# B&R Automation Studio project Nitto (part 16)

#### FB_GetNextCuttingSynPos.st
```iecst
(********************************************************************
 * COPYRIGHT -- Nitto
 ********************************************************************
 * Programm: MAIN
 * Datei: FB_GetNextCuttingSynPos.st
 * Autor: s_spilker
 * Erstellt: 9. November 2015
 ********************************************************************
 * Implementierung des Programms MAIN
 ********************************************************************)

(* TODO: Bitte Kommentar hier einfügen *)
FUNCTION_BLOCK FB_GetNextCuttingSynPos
// zu brmfmod die Funktion soll einen Rest der zwei Längen berechnen
// wenn die zwei Längen gelich sind (ausgenommen die Nachkommastellen fängt der Wert zu jittern (der Wert springt zwischen 0 und der Periodenlänge)

	periodLength :=	uData.general.periodLength;
	getMark(machineMaster := machineMaster, uData := uData, markpoints := markpoints, uAxis := uAxis, usercorrec := setCutOffset.setOffset_o);
//		IF period = 1 THEN //nur für Testzwecke
//		IF moduloBeforePosition > 0 THEN
//			IF moduloBeforePosition > periodLength THEN
//				correctionTotal1 := fmod(moduloBeforePosition, periodLength);
//				syncDataBefore.correctionNoLimit := correctionTotal1;
//				correctionTotalInt := 1;
//			ELSIF moduloBeforePosition < periodLength THEN
//				syncDataBefore.correctionNoLimit := (periodLength - moduloBeforePosition);
//				correctionTotalInt := 2;
//			END_IF
//		ELSIF 	moduloBeforePosition < 0 THEN
//			IF moduloBeforePosition < - periodLength THEN
//				correctionTotal1 := fmod(moduloBeforePosition, periodLength);
//				syncDataBefore.correctionNoLimit :=  correctionTotal1;
//				correctionTotalInt := 3;
//			ELSIF moduloBeforePosition > - periodLength THEN
//				syncDataBefore.correctionNoLimit := moduloBeforePosition + periodLength;
//				correctionTotalInt := 4;
//			END_IF
//
//		ELSIF moduloBeforePosition = periodLength THEN
//				syncDataBefore.correctionNoLimit := 0;
//				correctionTotalInt := 5;
//		END_IF
//	ELSIF period =	2 THEN
//		IF ABS ( moduloBeforePosition) > periodLength THEN
//			correctionTotal1 := fmod(ABS (moduloBeforePosition), periodLength);
//			syncDataBefore.correctionNoLimit := correctionTotal1 - periodLength;
//			correctionTotalInt := 6;
//		ELSIF ABS (moduloBeforePosition) < periodLength THEN
//			syncDataBefore.correctionNoLimit := correctionTotal1;
//			correctionTotalInt := 7;
//		END_IF
//	ELSIF period = 3 THEN
//			correctionTotal1 := fmod(moduloBeforePosition, periodLength);
//			IF correctionTotal1 > periodLength/2 THEN
//				syncDataBefore.correctionNoLimit := correctionTotal1 - periodLength;
//			ELSE
//				syncDataBefore.correctionNoLimit := correctionTotal1;
//			END_IF
//	ELSIF period =4 THEN
//			correctionTotal1 := fmod(ABS (moduloBeforePosition), periodLength);
//				IF correctionTotal1 > periodLength/2 THEN
//				syncDataBefore.correctionNoLimit := correctionTotal1 - periodLength;
//			ELSE
//				syncDataBefore.correctionNoLimit := correctionTotal1;
//			END_IF
//	ELSIF period = 5 THEN
//		correctionTotal1 := fmod(moduloBeforePosition, periodLength);
//	END_IF
//////permantes Lesen der Kurvenscheibenposition des Masters X-Achse 607, 512, 1067,
//	MC_BR_ReadCyclicPosition_1(Enable := TRUE, ParID:= 542, Axis := uAxis.AxisREF);//nur zu Testzwecken
	MC_BR_ReadCyclicPosition_0(Enable := TRUE, ParID:= 1075, Axis := uAxis.AxisREF);
//	moduloBeforePosition := MC_BR_ReadCyclicPosition_0.CyclicPosition.Integer - uData.general.periodLength;
	moduloBeforePosition := MC_BR_ReadCyclicPosition_0.CyclicPosition.Real - uData.general.periodLength;
	IF uData.recipe.mode = CONST.CUTTINGUNIT.MODEs.FREE_RUN THEN
		//für einen Rundenzähler
		countRtrig();
		IF MC_BR_ReadCyclicPosition_0.CyclicPosition.Real < 5000 THEN
			countRtrig.CLK := TRUE;
		END_IF
		IF countRtrig.Q	THEN
			syncDataBefore.markIndx := syncDataBefore.markIndx + 1;
			syncDataBefore.correctionNoLimit :=	- setCutOffset.setOffset_o;
		END_IF
		IF MC_BR_ReadCyclicPosition_0.CyclicPosition.Real > 10000 THEN
			countRtrig.CLK := FALSE;
		END_IF
	ELSIF uData.recipe.mode = CONST.CUTTINGUNIT.MODEs.SYNC_RUN OR uData.recipe.mode = CONST.CUTTINGUNIT.MODEs.CROSS_CUT THEN
			IF 	markpoints.ProbeCounter <> tmpcounter  OR trigger THEN
	//			correctionTotal := getMark.diffToUnitBefore - MC_BR_ReadCyclicPosition_0.CyclicPosition.Real;
				correctionTmp	:= fmod(getMark.diffToUnitBefore, uData.general.periodLength);
	//			correctionTotal := getMark.diffToUnitBefore - moduloBeforePosition;////03.11
				correctionTotal := correctionTmp - moduloBeforePosition;
				syncDataBefore.correctionNoLimit := correctionTotal;
				trigger := FALSE;
				syncDataBefore.markIndx := markpoints.ProbeCounter;
				tmpcounter := markpoints.ProbeCounter;
			ELSIF markpoints.MissedTriggers <> period THEN
				syncDataBefore.correctionNoLimit := correctionTotal;// LETZTEN BEKQNNTN WERT ALS KORREKTUR VORGEBEN
				period := markpoints.MissedTriggers;
			END_IF
	END_IF

END_FUNCTION_BLOCK
```

#### FB_CreateCamTable.st
```iecst
(********************************************************************
 * COPYRIGHT -- Nitto
 ********************************************************************
 * Programm: MAIN
 * Datei: FB_CreateCamTable.st
 * Autor: s_spilker
 * Erstellt: 9. November 2015
 ********************************************************************
 * Implementierung des Programms MAIN
 ********************************************************************)

(* TODO: Bitte Kommentar hier einfügen *)
FUNCTION_BLOCK FB_CreateCamTable
	CASE state OF

		STATE_READY://0
			IF createCam THEN
				(*	createCam:=FALSE;*)
				err(reset := TRUE);
				IF  data.recipe.tool.numberToolSegments = 1 OR data.recipe.tool.numberToolSegments = 0 OR data.recipe.mode = CONST.CUTTINGUNIT.MODEs.FREE_RUN THEN
					idx := 0;
					state:=STATE_CALCULATE_CAM1;
				ELSIF data.recipe.tool.numberToolSegments > 1 AND data.recipe.mode = CONST.CUTTINGUNIT.MODEs.SYNC_RUN THEN
					idx := 0;
					jdx := 0;
					state:=STATE_CALCULATE_CAM2;
				END_IF
			ELSE
				done:=FALSE;
			END_IF
		(*********************************************)
		STATE_CALCULATE_CAM1://1  (*calculate cam from sections*)
			(*bestimmung der Eigenschaften der Stützpunkte. Es können bis zu 64 Stützpunkte angelegt werden*)
			IF data.recipe.mode = CONST.CUTTINGUNIT.MODEs.FREE_RUN THEN // beim Freilauf wird Insetting auf ganzen Umfang bezogen
				CamSections.Section[0].MasterPosition	:=0;
				CamSections.Section[0].SlavePosition	:=0;
				CamSections.Section[0].FirstDerivative 	:= 1; (* Laut Ronny bei 1 wird die Geschwind. vom Master übernommen'*)
				CamSections.Section[0].SecondDerivative := 0;
				CamSections.Section[0].Mode 			:= mcABSOLUTE;(*mcRELATIVE;*)
				CamSections.Section[0].Type 			:= mc5TH_ORDER_POLYNOMIAL;

				CamSections.Section[1].MasterPosition 	:= scalePerimeter.realperimeter;// da das Werkzeug 1 zu 1 laufen soll
				CamSections.Section[1].SlavePosition 	:= scalePerimeter.realperimeter;
				CamSections.Section[1].FirstDerivative 	:= 1;
				CamSections.Section[1].SecondDerivative	:= 0;
				CamSections.Section[1].Mode 			:= mcABSOLUTE;  (*mcRELATIVE;*)
				CamSections.Section[1].Type 			:= mcLAST_POINT;(* mc5TH_ORDER_POLYNOMIAL;*)
				idx := 2;
				maxIdx := 64;
				WHILE idx < maxIdx -1 DO // falls bereits Stützpunkte vorhanden, alle löschen
					CamSections.Section[idx].MasterPosition		:= 0;
					CamSections.Section[idx].SlavePosition 		:= 0;
					CamSections.Section[idx].FirstDerivative 	:= 0; (* Laut Ronny bei 1 wird die Geschwind. vom Master übernommen'*)
					CamSections.Section[idx].SecondDerivative 	:= 0;
					CamSections.Section[idx].Mode 				:= 0;
					CamSections.Section[idx].Type 				:= 0;///mc5TH_ORDER_POLYNOMIAL;
					idx := idx +1;
				END_WHILE

				state:= STATE_CALC_CAM_FROM_SECTIONS;

			ELSIF data.recipe.mode = CONST.CUTTINGUNIT.MODEs.SYNC_RUN OR data.recipe.mode = CONST.CUTTINGUNIT.MODEs.CROSS_CUT THEN

				IF   data.recipe.tool.cutEndPosition > data.recipe.tool.cutStartPosition AND data.recipe.tool.cutEndPosition > 0 THEN
					//Kurvenscheibe mit einer synchnoner Strecke
					CamSections.Section[0].MasterPosition:=0;
					CamSections.Section[0].SlavePosition:=0;
					CamSections.Section[0].FirstDerivative := 1; (* Laut Ronny bei 1 wird die Geschwind. vom Master übernommen'*)
					CamSections.Section[0].SecondDerivative := 0;
					CamSections.Section[0].Mode := mcABSOLUTE;(*mcRELATIVE;*)
					CamSections.Section[0].Type := mcSTRAIGHT_LINE;///mc5TH_ORDER_POLYNOMIAL;
					// Ende der Kurvenscheibenstrecke mit einem automatischen Ausgleich und Anfang des Ausgleichs
					CamSections.Section[1].MasterPosition:= data.recipe.tool.cutEndPosition;
					CamSections.Section[1].SlavePosition:=data.recipe.tool.cutEndPosition;
					CamSections.Section[1].FirstDerivative := 1; (* Laut Ronny bei 1 wird die Geschwind. vom Master übernommen'*)
					CamSections.Section[1].SecondDerivative := 0;
					CamSections.Section[1].Mode := mcABSOLUTE;(*mcRELATIVE;*)
					CamSections.Section[1].Type := mc5TH_ORDER_POLYNOMIAL;//mcHARMONIC_COMBINATION ;
					//
					CamSections.Section[2].MasterPosition :=data.general.periodLength;
					CamSections.Section[2].SlavePosition := scalePerimeter.realperimeter;
					CamSections.Section[2].FirstDerivative := 1;
					CamSections.Section[2].SecondDerivative:= 0;
					CamSections.Section[2].Mode := mcABSOLUTE;  (*mcRELATIVE;*)
					CamSections.Section[2].Type := mcLAST_POINT;(* mc5TH_ORDER_POLYNOMIAL;*)

					idx := 3;
					maxIdx := 64;
					WHILE idx < maxIdx -1 DO // falls bereits Stützpunkte vorhanden, alle löschen

						CamSections.Section[idx].MasterPosition		:= 0;
						CamSections.Section[idx].SlavePosition 		:= 0;
						CamSections.Section[idx].FirstDerivative 	:= 0; (* Laut Ronny bei 1 wird die Geschwind. vom Master übernommen'*)
						CamSections.Section[idx].SecondDerivative 	:= 0;
						CamSections.Section[idx].Mode 				:= 0;
						CamSections.Section[idx].Type 				:= 0;///mc5TH_ORDER_POLYNOMIAL;
						idx := idx +1;
					END_WHILE
					state:= STATE_CALC_CAM_FROM_SECTIONS;

				ELSIF  data.recipe.tool.cutEndPosition = 0 OR data.recipe.tool.cutEndPosition = scalePerimeter.realperimeter THEN
					CamSections.Section[0].MasterPosition:=0;
					CamSections.Section[0].SlavePosition:=0;
					CamSections.Section[0].FirstDerivative := 1; (* Laut Ronny bei 1 wird die Geschwind. vom Master übernommen'*)
					CamSections.Section[0].SecondDerivative := 0;
					CamSections.Section[0].Mode := mcABSOLUTE;(*mcRELATIVE;*)
					CamSections.Section[0].Type := mc5TH_ORDER_POLYNOMIAL;

					CamSections.Section[1].MasterPosition :=data.general.periodLength;
					CamSections.Section[1].SlavePosition := scalePerimeter.realperimeter;
					CamSections.Section[1].FirstDerivative := 1;
					CamSections.Section[1].SecondDerivative:= 0;
					CamSections.Section[1].Mode := mcABSOLUTE;  (*mcRELATIVE;*)
					CamSections.Section[1].Type := mcLAST_POINT;(* mc5TH_ORDER_POLYNOMIAL;*)
					idx := 2;
					maxIdx := 64;
					WHILE idx < maxIdx -1 DO // falls bereits Stützpunkte vorhanden, alle löschen
						CamSections.Section[idx].MasterPosition		:= 0;
						CamSections.Section[idx].SlavePosition 		:= 0;
						CamSections.Section[idx].FirstDerivative 	:= 0; (* Laut Ronny bei 1 wird die Geschwind. vom Master übernommen'*)
						CamSections.Section[idx].SecondDerivative 	:= 0;
						CamSections.Section[idx].Mode 				:= 0;
						CamSections.Section[idx].Type 				:= 0;///mc5TH_ORDER_POLYNOMIAL;
						idx := idx +1;
					END_WHILE
					state:= STATE_CALC_CAM_FROM_SECTIONS;
				END_IF
			ELSIF data.recipe.tool.cutEndPosition < data.recipe.tool.cutStartPosition THEN
				err.set := TRUE;
				err.state := state;
				err.text := 'Synchronerbereich ist größer als Nutzen';
				err.fnc := 'FB_Camtable';
				err.id := MC_BR_CalcCamFromSections_0.ErrorID;
				state:=STATE_ERROR;
			END_IF

		STATE_CALCULATE_CAM2://1  (*calculate cam from sections*)
			(*Bestimmung der Eigenschaften der Stützpunkte. Es können bis zu 64 Stützpunkte angelegt werden*)
			IF data.recipe.tool.numberToolSegments > 1 AND  data.recipe.tool.numberToolSegments <= 12 THEN
				partOfPerimeter := scalePerimeter.realperimeter/data.recipe.tool.numberToolSegments;  //Anzahl der Kurvenstücken
				maxIdx			:= data.recipe.tool.numberToolSegments *2;
			ELSE
				partOfPerimeter := scalePerimeter.realperimeter;
			END_IF

			IF data.recipe.tool.cutEndPosition < partOfPerimeter  THEN
				CamSections.Section[maxIdx].MasterPosition	:= scalePerimeter.realperimeter;
				CamSections.Section[maxIdx].SlavePosition	:= scalePerimeter.realperimeter;
				CamSections.Section[maxIdx].FirstDerivative := 1; (* Laut Ronny bei 1 wird die Geschwind. vom Master übernommen'*)
				CamSections.Section[maxIdx].SecondDerivative:= 0;
				CamSections.Section[maxIdx].Mode 			:= mcABSOLUTE;
				CamSections.Section[maxIdx].Type 			:= mcLAST_POINT;
				WHILE idx < maxIdx -1 DO //jeden zweiten Stützpunkt, gerade Zahl
					CamSections.Section[idx].MasterPosition		:= partOfPerimeter * jdx;
					CamSections.Section[idx].SlavePosition 		:= partOfPerimeter * jdx;
					CamSections.Section[idx].FirstDerivative 	:= 1;
					CamSections.Section[idx].SecondDerivative 	:= 0;
					CamSections.Section[idx].Mode 				:= mcABSOLUTE;
					CamSections.Section[idx].Type 				:= mcSTRAIGHT_LINE; //mc5TH_ORDER_POLYNOMIAL;
					idx := idx + 2;
					jdx := jdx + 1;
				END_WHILE

				idx := 1;
				jdx := 0;
				WHILE idx < maxIdx DO//jede ungeraden Stützpuknt
					CamSections.Section[idx].MasterPosition		:= partOfPerimeter * jdx + data.recipe.tool.cutEndPosition;
					CamSections.Section[idx].SlavePosition 		:= partOfPerimeter * jdx + data.recipe.tool.cutEndPosition;
					CamSections.Section[idx].FirstDerivative 	:= 1; (* Laut Ronny bei 1 wird die Geschwind. vom Master übernommen'*)
					CamSections.Section[idx].SecondDerivative 	:= 0;
					CamSections.Section[idx].Mode 				:= mcABSOLUTE;
					CamSections.Section[idx].Type 				:= mc5TH_ORDER_POLYNOMIAL;///
					idx := idx + 2;
					jdx := jdx + 1;
				END_WHILE
				state:= STATE_CALC_CAM_FROM_SECTIONS;
			ELSE
				err.set := TRUE;
				err.state := state;
				err.text := 'Synchronerbereich ist größer als Nutzen';
				err.fnc := 'FB_Camtable';
				err.id := MC_BR_CalcCamFromSections_0.ErrorID;
				state:=STATE_ERROR;
			END_IF

		STATE_CALC_CAM_FROM_SECTIONS://2 //hier werden einzelne Punkte die in STATE_CALCULATE_CAM angelegt wurden sind als eine Stätige Kurve zusammen gesetzt
			idx := 0;
			MC_BR_CalcCamFromSections_0.Execute:= TRUE;
			MC_BR_CalcCamFromSections_0.DataAddress:=ADR(CamSections);
			MC_BR_CalcCamFromSections_0.CamProfileAddress:=ADR(MC_CAMPROFILE_TYP_0);
			MC_BR_CalcCamFromSections_0();

			IF MC_BR_CalcCamFromSections_0.Done THEN
				MC_BR_CalcCamFromSections_0.Execute:= FALSE;
				(*state:=STATE_READY;*)
				state := STATE_SAVE_CAM_PROFILE;
			ELSIF MC_BR_CalcCamFromSections_0.Error THEN
				err.set := TRUE;
				err.state:= state;
				err.text :='MC_BR_CalcCamFromSections_0';
				err.fnc := 'FB_Camtable';
				err.id := MC_BR_CalcCamFromSections_0.ErrorID;
				axis1ErrorID:= MC_BR_CalcCamFromSections_0.ErrorID;
				MC_BR_CalcCamFromSections_0.Execute:=0;
				state:=STATE_ERROR;
			END_IF

		STATE_SAVE_CAM_PROFILE:  //3 schreibe die Kurvenscheibe in das NC-Kurvenscheiben-Datenmodul
			MC_BR_CalcCamFromSections_0(); //noch einen Zyklus aufrufen

			MC_BR_SaveCamProfileObj_0.Execute			:= TRUE;
			MC_BR_SaveCamProfileObj_0.DataObjectName	:= Name; //'TestCam'; //Sehr wichtig der Name darf nicht größer als 12 Zeichen sein
			// Wie es bei B&R üblich ist, steht es explizit nirgendswo geschrieben. Nach mühsamen Test hat sich es gezeigt.
			MC_BR_SaveCamProfileObj_0.DataAddress		:= ADR(MC_CAMPROFILE_TYP_0);
			MC_BR_SaveCamProfileObj_0.DataObjectVersion	:= 1000;

			MC_BR_SaveCamProfileObj_0();

			IF MC_BR_SaveCamProfileObj_0.Done  THEN
				MC_BR_SaveCamProfileObj_0.Execute	:= FALSE;
				state:=STATE_DOWNLOAD_CAMPROFILEDATA;
			ELSIF MC_BR_SaveCamProfileObj_0.Error THEN
				err.set := TRUE;
				err.state := state;
				err.text := 'MC_BR_SaveCamProfileObj_0';
				err.fnc := 'FB_Camtable';
				err.id := MC_BR_SaveCamProfileObj_0.ErrorID;
				state := STATE_ERROR;
			END_IF

		STATE_DOWNLOAD_CAMPROFILEDATA://4 übertrage die Daten vom NC-Kurvenscheiben-Datenmodul auf den Antrieb
			(* zulässiger  an index for cam (1-14)*)
			MC_BR_SaveCamProfileObj_0();

			MC_BR_DownloadCamProfileObj_0.Execute 		:= TRUE;
			MC_BR_DownloadCamProfileObj_0.DataObjectName:= Name;
			MC_BR_DownloadCamProfileObj_0.Index			:= index;
			MC_BR_DownloadCamProfileObj_0.Periodic		:= mcPERIODIC;

			MC_BR_DownloadCamProfileObj_0(Axis := AxisREF);

			IF MC_BR_DownloadCamProfileObj_0.Done THEN
				MC_BR_DownloadCamProfileObj_0.Execute := FALSE;
				state :=  STATE_CAMTABLE_SEL;
			ELSIF MC_BR_DownloadCamProfileObj_0.Error THEN
				err.set := TRUE;
				err.state :=  state;
				err.text := 'MC_BR_DownloadCamProfileObj_0';
				err.fnc := 'FB_Camtable';
				err.id := MC_BR_DownloadCamProfileObj_0.ErrorID;
				state := STATE_ERROR;
			END_IF

		STATE_CAMTABLE_SEL: //5 wählt eine vordefinierte Kurvensscheibe ausfür den FB MC_CamIn.
			MC_BR_DownloadCamProfileObj_0(Axis := AxisREF);

			MC_CamTableSelect_0.CamTable := Name;
			MC_CamTableSelect_0.Periodic := mcPERIODIC; //periodische Achse
			MC_CamTableSelect_0.Execute := TRUE;
			MC_CamTableSelect_0(Master := MasterAxisREF, Slave := AxisREF);
			IF MC_CamTableSelect_0.Done AND MC_CamTableSelect_0.CamTableID > 0 THEN
				camTableID := MC_CamTableSelect_0.CamTableID; //zwischenspeichern weil beim nächsten Aufruf die CamTableID auf 0 gesetzt wird
				MC_CamTableSelect_0.Execute := FALSE;
				(*	done:=TRUE;*)
				//	createCam:=FALSE;//16.04.15 wird aus dem Config auf rückgesetzt.
				state := STATE_COMPLETED;
			ELSIF MC_CamTableSelect_0.Error THEN
				err(set := TRUE, text := 'MC_CamTableSelect_0', fnc := 'FB_Camtable', id := MC_CamTableSelect_0.ErrorID);
				state := STATE_ERROR;
			END_IF

		STATE_COMPLETED://10 FB werden noch mal aufgerufen um den Ausgang Done auf false zu setzten
			MC_BR_CalcCamFromSections_0(Execute := FALSE);
			MC_BR_SaveCamProfileObj_0(Execute := FALSE);
			MC_BR_DownloadCamProfileObj_0(Execute := FALSE);
			MC_CamTableSelect_0(Master := MasterAxisREF, Slave := AxisREF, Execute := FALSE);
			IF data.recipe.mode = CONST.CUTTINGUNIT.MODEs.FREE_RUN THEN
				IF MC_CAMPROFILE_TYP_0.MasterPeriod = REAL_TO_DINT(scalePerimeter.realperimeter) AND MC_CAMPROFILE_TYP_0.SlavePeriod = REAL_TO_DINT (scalePerimeter.realperimeter) THEN
					done:=TRUE;
					state := STATE_READY;
				END_IF
			ELSIF data.recipe.mode = CONST.CUTTINGUNIT.MODEs.SYNC_RUN THEN
				IF (*MC_CAMPROFILE_TYP_0.MasterPeriod >= REAL_TO_DINT(scalePerimeter.realperimeter) AND *)MC_CAMPROFILE_TYP_0.SlavePeriod = REAL_TO_DINT (scalePerimeter.realperimeter) THEN
					done:=TRUE;
					state := STATE_READY;
				END_IF
			END_IF

		STATE_ERROR:
			createCam:=FALSE;
			err();
			state:=STATE_READY;

	END_CASE
END_FUNCTION_BLOCK
```

#### FB_MARK_POSITION.st
```iecst
(********************************************************************
 * COPYRIGHT -- Nitto
 ********************************************************************
 * Programm: MAIN
 * Datei: FB_MARK_POSITION.st
 * Autor: s_spilker
 * Erstellt: 9. November 2015
 ********************************************************************
 * Implementierung des Programms MAIN
 ********************************************************************)

(* TODO: Bitte Kommentar hier einfügen *)
FUNCTION_BLOCK FB_MARK_POSITION
END_FUNCTION_BLOCK
```

#### Package Logical/MainMachineCtrl/MAIN/Longcutter - Paket

#### ac_manualLongCut.st
```iecst
(********************************************************************
 * COPYRIGHT -- Microsoft
 ********************************************************************
 * Programm: MAIN
 * Datei: acmanualLongCut.st
 * Autor: awalz
 * Erstellt: 30. Juni 2014
 ********************************************************************
 * Implementierung des Programms MAIN
 ********************************************************************)

(* Fügt eine neue Aktion zum IEC Programm oder Bibliothek *)
ACTION ac_manualLongCut:
		axis.ctrl();
		config( machineMasterCtrl := machineMaster, axis := axis, status := status);
	CASE state OF
	ST_IDLE:
		IF config.busy OR config.cmd <> CONST.CUTTINGUNIT.CMDs.NO_CMD THEN
			config(cmd := CONST.CUTTINGUNIT.CMDs.NO_CMD, machineMasterCtrl := machineMaster, axis := axis, status := status);
		ELSIF manualFirst  OR mode <> status.mode (*OR NewData *)THEN
			IF NOT status.isCoupled AND mode = CONST.UNITMODEs.ENABLE (*AND axis.ctrl.MC_ReadStatus_0.Disabled *)THEN
				axis.ctrl(cmd:= CONST.AXIS.POWER_ON);
				IF axis.ctrl.MC_ReadStatus_0.StandStill THEN
					status(mode := mode,axisState := axis.ctrl.MC_ReadStatus_0 );
					config(cmd := CONST.CUTTINGUNIT.CMDs.CPL_ON, machineMasterCtrl := machineMaster, axis := axis, status := status);
					state := ST_CPL_WAIT;
				END_IF
			ELSIF mode = CONST.UNITMODEs.DISABLE AND status.isCoupled THEN
				status(mode := mode,axisState := axis.ctrl.MC_ReadStatus_0 );
				config(cmd := CONST.CUTTINGUNIT.CMDs.CPL_OFF, machineMasterCtrl := machineMaster, axis := axis, status := status);
				state := ST_CPL_WAIT;
//			ELSIF	mode = CONST.UNITMODEs.AXIS_OFF THEN
//				status(mode := mode,axisState := axis.ctrl.MC_ReadStatus_0 );
//				axis.ctrl(cmd:= CONST.AXIS.POWER_OFF);
//				status.isCoupled := FALSE;
//				state := ST_AXIS_OFF;
//			ELSIF	mode = CONST.UNITMODEs.DISABLE AND axis.ctrl.MC_ReadStatus_0.Disabled THEN
//				status(mode := mode,axisState := axis.ctrl.MC_ReadStatus_0 );
//				status.isCoupled := FALSE;
//				axis.ctrl(cmd:= CONST.AXIS.POWER_ON);
//				state := ST_AXIS_ON;
////////////////////////
			ELSIF cmdCtrl.value = CONST.CUTTINGUNIT.CMDs.MOVEFW (*OR cmdCtrl.value = CONST.CUTTINGUNIT.CMDs.MOVEBW*) THEN
				cmdStatus(set := TRUE, value := cmdCtrl.value);
				busy := TRUE;
				state := ST_MOVE_START;
//////////////////////////
			ELSE
				NewData := FALSE;
				manualFirst := FALSE;
			END_IF
		ELSIF cmdCtrl.value <> CONST.CUTTINGUNIT.CMDs.NO_CMD THEN
			cmdStatus(set := TRUE, value := cmdCtrl.value);
			busy := TRUE;
			state := ST_FUNCTION_START;
		END_IF

	ST_CPL_WAIT:
		config( machineMasterCtrl := machineMaster, axis := axis, status := status);
		(*status(mode := mode);*)
		IF NOT config.busy THEN
			IF config.err.flag THEN
				err := config.err;
				err.state := state;
				state := ST_ERROR;
			ELSE
				manualFirst := FALSE;
				axis.setGearRatio.init := TRUE;  // OKrebs 09.12.15
				state := ST_IDLE;
			END_IF
			config(cmd := CONST.CUTTINGUNIT.CMDs.NO_CMD, machineMasterCtrl := machineMaster, axis := axis, status := status );
		END_IF

	ST_FUNCTION_START:
		IF config.busy OR config.cmd <> CONST.CUTTINGUNIT.CMDs.NO_CMD THEN
			config(cmd := CONST.CUTTINGUNIT.CMDs.NO_CMD, machineMasterCtrl := machineMaster, axis := axis, status := status);
		ELSE
			config(cmd := cmdStatus.value, machineMasterCtrl := machineMaster, axis := axis, status := status);
			state := ST_FUNCTION;
		END_IF

	ST_FUNCTION:
		config( machineMasterCtrl := machineMaster, axis := axis, status := status);
		IF NOT config.busy THEN
			IF config.err.flag THEN
				err := config.err;
				err.state := state;
			END_IF
			config(cmd := CONST.CUTTINGUNIT.CMDs.NO_CMD, machineMasterCtrl := machineMaster, axis := axis, status := status );
			state := ST_FUNCTION_QUIT;
		END_IF
////12.08.14/////
	ST_MOVE_START:
			config(cmd := cmdStatus.value, machineMasterCtrl  := machineMaster, axis := axis, status := status);
			state := ST_MOVE;

	ST_MOVE:
//		config (machineMaster := machineMaster, axis := axis, status := status, data := data, IOs := IOs, powerbridge := powerbridge,
//				scalePerimeter := scalePerimeter, getNextCuttPos := getNextCuttPos);
		IF cmdCtrl.value = CONST.CUTTINGUNIT.CMDs.NO_CMD THEN
			config(cmd := CONST.CUTTINGUNIT.CMDs.NO_CMD, machineMasterCtrl := machineMaster, axis := axis, status := status);
			state := ST_MOVE_QUIT;

		ELSE
			config(cmd := cmdStatus.value, machineMasterCtrl := machineMaster, axis := axis, status := status);
		END_IF

	ST_MOVE_QUIT:
		config(cmd := CONST.CUTTINGUNIT.CMDs.NO_CMD, machineMasterCtrl := machineMaster, axis := axis, status := status);
		IF NOT config.busy THEN
			busy := FALSE;
			cmdStatus(set := TRUE, value := CONST.CUTTINGUNIT.CMDs.NO_CMD);
			state := ST_IDLE;
		END_IF

////////////////////////////////
	ST_AXIS_OFF:
	(*	status(mode := mode);*)
		IF mode <> CONST.UNITMODEs.AXIS_OFF THEN
			state := ST_IDLE;
		END_IF
	ST_AXIS_ON:
	(*	status(mode := mode);*)
		IF mode <> CONST.UNITMODEs.DISABLE THEN
			state := ST_IDLE;
		END_IF

	ST_FUNCTION_QUIT:
		busy := FALSE;
		IF cmdCtrl.value = CONST.CUTTINGUNIT.CMDs.NO_CMD THEN
			cmdStatus(set :=TRUE, value := CONST.CUTTINGUNIT.CMDs.NO_CMD);
			state := ST_IDLE;
		END_IF

	ST_ERROR:
		err.flag := TRUE;
		busy := FALSE;
		IF BetrCtrl.value <> CONST.MACHINEMODES.MANUAL THEN
			state := ST_IDLE;
			err(reset := TRUE);
			busy := TRUE;
			StateCtrl := CTRL_MANUAL_AFTER;
		END_IF
	END_CASE

	(*axis.calcGearRatio(enable := ( data.torqueCtrlOn  AND axis.ctrl.ref.Status.Coupled), axisRef := axis.ctrl.ref, zugRegelWert := zugRegelWert);*)
END_ACTION
```

#### FB_LongcutterCtrl.st
```iecst
(********************************************************************
 * COPYRIGHT -- Microsoft
 ********************************************************************
 * Programm: MAIN
 * Datei: FB_LongcutterCtrl.st
 * Autor: awalz
 * Erstellt: 29. Juni 2014
 ********************************************************************
 * Implementierung des Programms MAIN
 ********************************************************************)

(* TODO: Bitte Kommentar hier einfügen *)
FUNCTION_BLOCK FB_LongcutterCtrl
	axis.ctrl();
	cutterUp(clk := clk, );(*cutterUp.enable wird dierekt vom EIngang 202A3Input6 geschaltet*)
	discmovesupp(clk := clk);
	movebutton(clk := clk);
	webclamp(clk := clk);
	status(axisState := axis.ctrl.MC_ReadStatus_0);
	status.ready := axis.ctrl.MC_ReadStatus_0.SynchronizedMotion;
	emcy_inputs();
	IF emcy_inputs.EMCY_Door1 THEN
		emcy_inputs.EMCY_DoorsClosed := TRUE;
	ELSE
		emcy_inputs.EMCY_DoorsClosed := FALSE;

	END_IF
	chkStatus(setMode := mode, status := status);
	axis.setGearRatio(limitvisuneg := -20, limitvisupos := 50, limitrationeg := 800, limitratiopos := 1500);
	IF machineMaster.MC_ReadStatus_0.ContinuousMotion THEN
		discmovesupp.toDown_o := FALSE;
	END_IF
//	IF axis.ctrl.MC_ReadStatus_0.SynchronizedMotion AND axis.setGearRatio.enable THEN
//
//
//	END_IF
	axis.cplOn.Execute := axis.setGearRatio.trigger OR movebutton.LDT.ftrig.Q OR axisCpl; // 25.07.18 // OKrebs

	axis.cplOn(RatioNumerator := axis.setGearRatio.ratioNumeratorOut,
				(*Execute := axis.setGearRatio.trigger, 25.07.18 OKrebs*) RatioDenominator := axis.setGearRatio.ratioDenominator,
					Acceleration := 40000, Deceleration := 40000);

//	IF  movebutton.LDT.ftrig.Q THEN	// 25.07.18 // OKrebs
//		axis.cplOn.Execute := TRUE; // 25.07.18 // OKrebs
//	END_IF							// 25.07.18 // OKrebs

////12.08.14 jog set commando  for Longcutter
	IF movebutton.LDT.button THEN
		cmdCtrl.value := CONST.CUTTINGUNIT.CMDs.MOVEFW;
	ELSIF movebutton.LDT.ftrig.Q THEN ////12.08.14 jog reset commando  for Longcutter
		cmdCtrl.value := CONST.CUTTINGUNIT.CMDs.NO_CMD;
	END_IF
////21.08.14 Um Achse zu reseten//
	IF cmdCtrl.value = CONST.CUTTINGUNIT.CMDs.RESET THEN
		axis.ctrl.cmd := CONST.AXIS.RESET;
	ELSIF cmdCtrl.value = CONST.CUTTINGUNIT.CMDs.NO_CMD THEN
		axis.ctrl.cmd := CONST.AXIS.NOACTION;
	END_IF
	status.axiserror := axis.ctrl.MC_ReadStatus_0.Errorstop;
	IF	mode = CONST.UNITMODEs.AXIS_OFF OR  NOT emcy_inputs.EMCY_Door1 THEN
				status(mode := mode,axisState := axis.ctrl.MC_ReadStatus_0 );
				axis.ctrl(cmd:= CONST.AXIS.POWER_OFF);
				status.isCoupled := FALSE;
				state := ST_AXIS_OFF;
	ELSIF	mode = CONST.UNITMODEs.ENABLE AND axis.ctrl.MC_ReadStatus_0.Disabled AND  emcy_inputs.EMCY_Door1 THEN
				status(mode := mode,axisState := axis.ctrl.MC_ReadStatus_0 );
				status.isCoupled := FALSE;
				axis.ctrl(cmd:= CONST.AXIS.POWER_ON);
				stateCPL := cpl_idle;
	ELSIF	mode = CONST.UNITMODEs.DISABLE AND NOT axis.ctrl.MC_ReadStatus_0.Disabled AND  emcy_inputs.EMCY_Door1 THEN
				status(mode := mode,axisState := axis.ctrl.MC_ReadStatus_0 );
				status.isCoupled := FALSE;
				axis.ctrl(cmd:= CONST.AXIS.POWER_ON);
				state := ST_AXIS_ON;
	END_IF
//////////////////////
	CASE stateCPL OF
		cpl_idle :
			IF axis.ctrl.MC_ReadStatus_0.StandStill THEN
				axisCpl := TRUE;
//				axis.cplOn.Execute := TRUE; // 25.07.18 // OKrebs
				stateCPL := clp_cpl;
			END_IF
		clp_cpl:
			axisCpl := FALSE;
				;
		END_CASE
	CASE StateCtrl OF
	CTRL_FIRST_START:
		busy := TRUE;
		StateCtrl := CTRL_EMERGENCYSTOP_BEFORE;

	CTRL_MANUAL_BEFORE:
		IF BetrCtrl.value = CONST.MACHINEMODES.MANUAL THEN
		(*	clamp.init(clk := clk);*)
			BetrStatus(set := TRUE, value := CONST.MACHINEMODES.MANUAL);
			chkStatus.enable := TRUE;
			err(reset := TRUE);
			busy := FALSE;
			timer(IN:= FALSE);
			state := ST_IDLE;
			manualFirst := TRUE;
			StateCtrl := CTRL_MANUAL;
//			axis.setGearRatio.init := TRUE;
		ELSIF BetrCtrl.value = CONST.MACHINEMODES.EMERGENCYSTOP THEN
			StateCtrl := CTRL_EMERGENCYSTOP_BEFORE;
		ELSIF BetrCtrl.value = CONST.MACHINEMODES.SAFETYSTOP THEN
			StateCtrl := CTRL_SAFETYSTOP_BEFORE;
		ELSIF BetrCtrl.value = CONST.MACHINEMODES.AUTOMATIC THEN
			StateCtrl := CTRL_AUTO_BEFORE;
		END_IF

	CTRL_MANUAL:
		IF BetrCtrl.value <> CONST.MACHINEMODES.MANUAL THEN
			err(reset := TRUE);
			busy := TRUE;
			StateCtrl := CTRL_MANUAL_AFTER;
//		ELSIF axis.ctrl.MC_ReadStatus_0.StandStill THEN
//			axis.ctrl.cmd := CONST.AXIS.START;
//				timer(IN := TRUE, PT := T#8s);
//				IF timer.Q THEN

			(*	END_IF*)
		ELSE
			ac_manualLongCut;
		END_IF

	CTRL_MANUAL_AFTER:
		timer(IN:= FALSE);
		chkStatus.enable := FALSE;
		axis.ctrl.cmd := CONST.AXIS.NOACTION;
		ac_setStateAfterPB;

	CTRL_AUTO_BEFORE:
		IF BetrCtrl.value = CONST.MACHINEMODES.AUTOMATIC THEN
		BetrStatus(set := TRUE, value := CONST.MACHINEMODES.AUTOMATIC);
			(*clamp.init(clk := clk);*)
			err(reset := TRUE);
			chkStatus.enable := TRUE;
			busy := FALSE;
			state := ST_IDLE;
			StateCtrl := CTRL_AUTO;
		ELSIF BetrCtrl.value = CONST.MACHINEMODES.EMERGENCYSTOP THEN
			StateCtrl := CTRL_EMERGENCYSTOP_BEFORE;
		ELSIF BetrCtrl.value = CONST.MACHINEMODES.SAFETYSTOP THEN
			StateCtrl := CTRL_SAFETYSTOP_BEFORE;
		ELSIF BetrCtrl.value = CONST.MACHINEMODES.MANUAL THEN
			StateCtrl := CTRL_MANUAL_BEFORE;
		END_IF

	(* ******************************** *)
	(* *********** AUTO *************** *)
	(* ******************************** *)
	CTRL_AUTO:
		IF BetrCtrl.value <> CONST.MACHINEMODES.AUTOMATIC THEN
			err(reset := TRUE);
			busy := TRUE;
			StateCtrl := CTRL_AUTO_AFTER;
		ELSE
			;(*ac_automatic();*)
		END_IF

	CTRL_AUTO_AFTER:
		chkStatus.enable := FALSE;
		state := ST_IDLE;
		ac_setStateAfterPB;

	CTRL_STOP_BEFORE:
		IF BetrCtrl.value = CONST.MACHINEMODES.EMERGENCYSTOP THEN
			StateCtrl := CTRL_EMERGENCYSTOP_BEFORE;
		ELSIF BetrCtrl.value = CONST.MACHINEMODES.SAFETYSTOP THEN
			StateCtrl := CTRL_SAFETYSTOP_BEFORE;
		ELSE
			state := ST_IDLE;
			StateCtrl := CTRL_STOP;
		END_IF

	CTRL_STOP:
		IF BetrCtrl.value = CONST.MACHINEMODES.EMERGENCYSTOP THEN
			StateCtrl := CTRL_EMERGENCYSTOP_BEFORE;
		ELSIF BetrCtrl.value = CONST.MACHINEMODES.SAFETYSTOP THEN
			StateCtrl := CTRL_SAFETYSTOP_BEFORE;
		ELSE
			CASE state OF
			ST_IDLE:
				state := ST_QUIT;

			ST_QUIT:
				state := ST_IDLE;
				StateCtrl := CTRL_STOP_AFTER;
			END_CASE
		END_IF

	CTRL_STOP_AFTER:
		IF BetrCtrl.value = CONST.MACHINEMODES.EMERGENCYSTOP THEN
			StateCtrl := CTRL_EMERGENCYSTOP_BEFORE;
		ELSIF BetrCtrl.value = CONST.MACHINEMODES.SAFETYSTOP THEN
			StateCtrl := CTRL_SAFETYSTOP_BEFORE;
		ELSIF BetrCtrl.value = CONST.MACHINEMODES.MANUAL THEN
			StateCtrl := CTRL_MANUAL_BEFORE;
		ELSIF BetrCtrl.value = CONST.MACHINEMODES.AUTOMATIC THEN
			StateCtrl := CTRL_AUTO_BEFORE;
		END_IF

	CTRL_RESET_START:
		BetrStatus(set := TRUE,value := CONST.MACHINEMODES.RESET);
		IF BetrCtrl.value = CONST.MACHINEMODES.EMERGENCYSTOP THEN
			StateCtrl := CTRL_EMERGENCYSTOP_BEFORE;
		ELSIF BetrCtrl.value = CONST.MACHINEMODES.SAFETYSTOP THEN
			StateCtrl := CTRL_SAFETYSTOP_BEFORE;
		ELSE
			IF axis.ctrl.busy OR axis.ctrl.cmd <> CONST.AXIS.NOACTION  THEN
				axis.ctrl(cmd := CONST.AXIS.NOACTION);
//			ELSIF axis.ctrl.MC_ReadStatus_0.Disabled THEN
//				axis.ctrl(cmd := CONST.AXIS.RESET);
//				StateCtrl := CTRL_RESET;
			ELSE
				axis.ctrl(cmd := CONST.AXIS.RESET);
				StateCtrl := CTRL_RESET;
			END_IF
		END_IF

	CTRL_RESET:
		axis.ctrl();
		IF BetrCtrl.value = CONST.MACHINEMODES.EMERGENCYSTOP THEN
			StateCtrl := CTRL_EMERGENCYSTOP_BEFORE;
		ELSIF BetrCtrl.value = CONST.MACHINEMODES.SAFETYSTOP THEN
			StateCtrl := CTRL_SAFETYSTOP_BEFORE;
		ELSE
//			IF NOT axis.ctrl.busy THEN (* auskommentiert am 26.06..14*)
//				axis.ctrl(cmd := CONST.AXIS.NOACTION);
//				StateCtrl := CTRL_RESET_AFTER;
//			END_IF
//			cutterUp.buttomToggle.LDT.button := TRUE;
//			cutterUp(clk := clk );
			axis.ctrl(cmd := CONST.AXIS.POWER_OFF);
			StateCtrl := CTRL_RESET_AFTER;
		END_IF

	CTRL_RESET_AFTER:
		IF BetrCtrl.value = CONST.MACHINEMODES.RESET THEN
			busy := FALSE;
		ELSE
			busy := TRUE;
			cutterUp(clk := clk, init := TRUE);
			err(reset := TRUE);
			IF BetrCtrl.value = CONST.MACHINEMODES.EMERGENCYSTOP THEN
				StateCtrl := CTRL_EMERGENCYSTOP_BEFORE;
			ELSIF BetrCtrl.value = CONST.MACHINEMODES.SAFETYSTOP THEN
				StateCtrl := CTRL_SAFETYSTOP_BEFORE;
			ELSIF BetrCtrl.value = CONST.MACHINEMODES.SAFETYSTOP THEN
				StateCtrl := CTRL_SAFETYSTOP_BEFORE;
			ELSIF BetrCtrl.value = CONST.MACHINEMODES.MANUAL  AND safety.valid THEN
				supplydelay(IN:= TRUE, PT := T#8s);
				IF supplydelay.Q THEN
					axis.ctrl(cmd := CONST.AXIS.POWER_ON);
					busy := TRUE;
					supplydelay(IN:= FALSE);
					StateCtrl := CTRL_MANUAL_BEFORE;
				END_IF
			ELSIF BetrCtrl.value = CONST.MACHINEMODES.AUTOMATIC  AND safety.valid THEN
				supplydelay(IN:= TRUE, PT := T#8s);
				IF supplydelay.Q THEN
					axis.ctrl(cmd := CONST.AXIS.POWER_ON);
					busy := TRUE;
					supplydelay(IN:= FALSE);
					StateCtrl := CTRL_AUTO_BEFORE;
				END_IF
			END_IF
		END_IF

	CTRL_SAFETYSTOP_BEFORE:
		status.isCoupled := FALSE;
		status.ready := FALSE;
		IF BetrCtrl.value = CONST.MACHINEMODES.EMERGENCYSTOP THEN
			StateCtrl := CTRL_EMERGENCYSTOP_BEFORE;
		ELSE
			BetrStatus(set := TRUE,value := CONST.MACHINEMODES.SAFETYSTOP);
			state := ST_IDLE;
			manualFirst := FALSE;
			axis.ctrl.verzoegerung	:= CONST.AXIS.EMERGENCY_DECELERATION;
			axis.ctrl.cmd := CONST.AXIS.STOP;
			StateCtrl := CTRL_SAFETYSTOP;
		END_IF

	CTRL_SAFETYSTOP:
		IF BetrCtrl.value = CONST.MACHINEMODES.EMERGENCYSTOP THEN
			StateCtrl := CTRL_EMERGENCYSTOP_BEFORE;
		ELSE
			BetrStatus(set := TRUE,value := CONST.MACHINEMODES.SAFETYSTOP);
			IF axis.ctrl.MC_ReadStatus_0.StandStill THEN
				axis.ctrl.cmd := CONST.AXIS.POWER_OFF;
			ELSIF axis.ctrl.MC_ReadStatus_0.Disabled THEN
				axis.ctrl.cmd := CONST.AXIS.NOACTION;
				StateCtrl := CTRL_SAFETYSTOP_AFTER;
			END_IF

		END_IF

	CTRL_SAFETYSTOP_AFTER:
		busy := FALSE;
		manualFirst := TRUE;
		status.ready := FALSE;
		IF axis.ctrl.MC_ReadStatus_0.Errorstop THEN
			axis.ctrl.cmd := CONST.AXIS.RESET;
		END_IF
		IF BetrCtrl.value = CONST.MACHINEMODES.EMERGENCYSTOP THEN
			busy := TRUE;
			StateCtrl := CTRL_EMERGENCYSTOP_BEFORE;
		ELSIF BetrCtrl.value = CONST.MACHINEMODES.MANUAL  AND safety.valid THEN
				supplydelay(IN:= TRUE, PT := T#8s);
				IF supplydelay.Q THEN
					axis.ctrl(cmd := CONST.AXIS.POWER_ON);
					busy := TRUE;
					supplydelay(IN:= FALSE);
					StateCtrl := CTRL_MANUAL_BEFORE;
				END_IF
		ELSIF BetrCtrl.value = CONST.MACHINEMODES.AUTOMATIC  AND safety.valid THEN
				supplydelay(IN:= TRUE, PT := T#8s);
				IF supplydelay.Q THEN
					axis.ctrl(cmd := CONST.AXIS.POWER_ON);
					busy := TRUE;
					supplydelay(IN:= FALSE);
					StateCtrl := CTRL_AUTO_BEFORE;
				END_IF
		END_IF

	CTRL_EMERGENCYSTOP_BEFORE:
		status.isCoupled := FALSE;
		status.ready := FALSE;
		cutterUp(clk := clk, init := TRUE);
		IF  axis.ctrl.MC_ReadStatus_0.ContinuousMotion OR axis.ctrl.MC_ReadStatus_0.DiscreteMotion
			OR axis.ctrl.MC_ReadStatus_0.SynchronizedMotion THEN //alle Zustände in denen die Achse sich bewegen kann
			axis.ctrl.verzoegerung:= CONST.AXIS.EMERGENCY_DECELERATION; (*200m/min in 3 sek*); (* von 200m/min in 2 sek*)
			axis.ctrl.cmd := CONST.AXIS.STOP;
			state := ST_IDLE;
			StateCtrl := CTRL_EMERGENCYSTOP;
		ELSE //wenn die Maschine eingeschaltet wird
			axis.ctrl.cmd := CONST.AXIS.NOACTION;
			state := ST_IDLE;
			StateCtrl := CTRL_EMERGENCYSTOP;
		END_IF

	CTRL_EMERGENCYSTOP:
		status.isCoupled := FALSE;
		status.ready := FALSE;
		IF BetrCtrl.value = CONST.MACHINEMODES.EMERGENCYSTOP THEN
			IF axis.ctrl.MC_ReadStatus_0.StandStill THEN
				axis.ctrl.cmd := CONST.AXIS.POWER_OFF;
				busy := FALSE;
			ELSIF axis.ctrl.MC_ReadStatus_0.Disabled THEN
				axis.ctrl.cmd := CONST.AXIS.NOACTION;
				busy := FALSE;
			END_IF
		ELSE
			busy := TRUE;
			timer(IN := TRUE, PT := T#2s);
			StateCtrl := CTRL_EMERGENCYSTOP_AFTER;
		END_IF

	CTRL_EMERGENCYSTOP_AFTER:
		timer();
		IF BetrCtrl.value = CONST.MACHINEMODES.EMERGENCYSTOP THEN
			timer(IN := FALSE);
			BetrStatus(set := TRUE , value := CONST.MACHINEMODES.EMERGENCYSTOP);
			busy := FALSE;
			StateCtrl := CTRL_EMERGENCYSTOP;
		ELSIF timer.Q THEN
			timer(IN := FALSE);
			StateCtrl := CTRL_RESET_START;
		END_IF

	ELSE
		;
	END_CASE
	axis.ctrl.BasicControl.Parameter.Deceleration	:= 40000.0; //only for initialization
	axis.ctrl.BasicControl.Parameter.Acceleration	:= 40000.0;
END_FUNCTION_BLOCK
```

#### FB_LONGCUTTER.st
```iecst
(********************************************************************
 * COPYRIGHT -- Microsoft
 ********************************************************************
 * Programm: MAIN
 * Datei: FB_LONGCUTTER.st
 * Autor: awalz
 * Erstellt: 29. Juni 2014
 ********************************************************************
 * Implementierung des Programms MAIN
 ********************************************************************)

(* TODO: Bitte Kommentar hier einfügen *)
FUNCTION_BLOCK FB_LONGCUTTER
END_FUNCTION_BLOCK
```

#### Package Logical/MainMachineCtrl/MAIN/Conveyor - Neues leeres Paket

#### FB_CONVEYOR_AXIS.st
```iecst
(********************************************************************
 * COPYRIGHT -- Microsoft
 ********************************************************************
 * Programm: MAIN
 * Datei: FB_CONVEYOR.st
 * Autor: Awalz
 * Erstellt: 12. Mai 2014
 ********************************************************************
 * Implementierung des Programms MAIN
 ********************************************************************)

 (*<$Description$> TODO: Bitte Kommentar hier einzufügen </$Description$>*)
FUNCTION_BLOCK FB_CONVEYOR_AXIS
END_FUNCTION_BLOCK
```

#### ac_manualConv.st
```iecst
(********************************************************************
 * COPYRIGHT -- Microsoft
 ********************************************************************
 * Programm: MAIN
 * Datei: ac_manualConv.st
 * Autor: Awalz
 * Erstellt: 12. Mai 2014
 ********************************************************************
 * Implementierung des Programms MAIN
 ********************************************************************)

 (*<$Description$> Fügt eine neue Aktion zum IEC Programm oder Bibliothek </$Description$>*)
ACTION ac_manualConv:
//		axis.ctrl();
		config( machineMasterCtrl := machineMaster, axis := axis, status := status);
	CASE state OF
	ST_IDLE:
		IF config.busy OR config.cmd <> CONST.CUTTINGUNIT.CMDs.NO_CMD THEN
			config(cmd := CONST.CUTTINGUNIT.CMDs.NO_CMD, machineMasterCtrl := machineMaster, axis := axis, status := status);
		ELSIF manualFirst  OR mode <> status.mode (*OR NewData *)THEN
			IF NOT status.isCoupled AND mode = CONST.UNITMODEs.ENABLE (*18.03.15*) AND axis.ctrl.MC_ReadStatus_0.StandStill THEN
				config(cmd := CONST.CUTTINGUNIT.CMDs.CPL_ON, machineMasterCtrl := machineMaster, axis := axis, status := status);
				state := ST_CPL_WAIT;
			ELSIF mode <> CONST.UNITMODEs.ENABLE AND status.isCoupled THEN
				config(cmd := CONST.CUTTINGUNIT.CMDs.CPL_OFF, machineMasterCtrl := machineMaster, axis := axis, status := status);
				state := ST_CPL_WAIT;
			ELSE
				NewData := FALSE;
//				manualFirst := FALSE;
			END_IF
		ELSIF cmdCtrl.value <> CONST.CUTTINGUNIT.CMDs.NO_CMD THEN
			cmdStatus(set := TRUE, value := cmdCtrl.value);
			busy := TRUE;
				state := ST_FUNCTION_START;
		ELSIF axis.ctrl.MC_ReadStatus_0.Disabled AND mode = CONST.UNITMODEs.ENABLE THEN//18.03.15
			axis.ctrl.cmd := CONST.AXIS.POWER_ON;
		END_IF

	ST_CPL_WAIT:
		config( machineMasterCtrl := machineMaster, axis := axis, status := status);
		IF NOT config.busy AND  mode = CONST.UNITMODEs.ENABLE THEN//18.03.15
			IF config.err.flag THEN
				err := config.err;
				err.state := state;
				state := ST_ERROR;
			ELSE
				manualFirst := FALSE;
				axis.setGearRatio.init := TRUE;	// OKrebs 09.12.15
				state := ST_IDLE;
			END_IF
				config(cmd := CONST.CUTTINGUNIT.CMDs.NO_CMD, machineMasterCtrl := machineMaster, axis := axis, status := status );
		ELSIF mode <> CONST.UNITMODEs.ENABLE THEN
				state := ST_IDLE;
		END_IF

	ST_FUNCTION_START:
//		IF config.busy OR config.cmd <> CONST.CUTTINGUNIT.CMDs.NO_CMD THEN
//			config(cmd := CONST.CUTTINGUNIT.CMDs.NO_CMD, machineMasterCtrl := machineMaster, axis := axis, status := status);
//		ELSE
			config(cmd := cmdStatus.value, machineMasterCtrl := machineMaster, axis := axis, status := status);
			state := ST_FUNCTION;
//		END_IF

	ST_FUNCTION:
//		config( machineMasterCtrl := machineMaster, axis := axis, status := status);
//		IF NOT config.busy THEN
//			IF config.err.flag THEN
//				err := config.err;
//				err.state := state;
			//			END_IF
		IF cmdCtrl.value = CONST.CUTTINGUNIT.CMDs.NO_CMD THEN
			config(cmd := CONST.CUTTINGUNIT.CMDs.NO_CMD, machineMasterCtrl := machineMaster, axis := axis, status := status );
			state := ST_FUNCTION_QUIT;
		END_IF

	ST_FUNCTION_QUIT:
		busy := FALSE;
		IF cmdCtrl.value = CONST.CUTTINGUNIT.CMDs.NO_CMD THEN
			cmdStatus(set :=TRUE, value := CONST.CUTTINGUNIT.CMDs.NO_CMD);
			state := ST_IDLE;
		END_IF

	ST_ERROR:
		err.flag := TRUE;
		busy := FALSE;
		IF BetrCtrl.value <> CONST.MACHINEMODES.MANUAL THEN
			state := ST_IDLE;
			err(reset := TRUE);
			busy := TRUE;
			StateCtrl := CTRL_MANUAL_AFTER;
		END_IF
	END_CASE

	(*axis.calcGearRatio(enable := ( data.torqueCtrlOn  AND axis.ctrl.ref.Status.Coupled), axisRef := axis.ctrl.ref, zugRegelWert := zugRegelWert);*)
END_ACTION
```

#### FB_ConveyorCtrl.st
```iecst
(********************************************************************
 * COPYRIGHT -- Microsoft
 ********************************************************************
 * Programm: MAIN
 * Datei: FB_ConveyorCtrl.st
 * Autor: Awalz
 * Erstellt: 12. Mai 2014
 ********************************************************************
 * Implementierung des Programms MAIN
 ********************************************************************)

 (*<$Description$> TODO: Bitte Kommentar hier einzufügen </$Description$>*)
FUNCTION_BLOCK FB_ConveyorCtrl
	axis.ctrl();
//	mode := CONST.UNITMODEs.ENABLE;
	chkStatus(setMode := mode, status := status);
	(*axis.setGearRatio();*)
	axis.setGearRatio(limitvisuneg := -80, limitvisupos :=400(*700*), limitrationeg := 1000, limitratiopos := 5000);
	emcy_inputs();
	panel();
	counters();
	status(axisState := axis.ctrl.MC_ReadStatus_0);
	status.ready := axis.ctrl.MC_ReadStatus_0.SynchronizedMotion;
 //24.07.18 //OKrebs // Falls das Band sich nicht mehr manuell bewegen laesst
	IF (config.state = 40) AND visuReset AND config.busy THEN
		axis.MC_BR_Phasing_0.Enable := FALSE;
		config.state := 0;
		config.busy := FALSE;
	END_IF
/////////////////////////////////////
	IF axis.ctrl.MC_ReadStatus_0.Errorstop AND panel.LDTRESET.LDT.button THEN
		axis.ctrl.cmd := CONST.AXIS.RESET;
		status.isCoupled := FALSE; // OKrebs // 24.07.18
		manualFirst	:= TRUE; // OKrebs // 24.07.18
	ELSIF axis.ctrl.MC_ReadStatus_0.Disabled AND panel.LDTRESET.LDT.ftrig.Q AND cmdCtrl.value = CONST.AXIS.NOACTION THEN
		axis.ctrl.cmd := CONST.AXIS.NOACTION;
	END_IF

	IF (*axis.ctrl.MC_ReadStatus_0.SynchronizedMotion AND*) axis.setGearRatio.enable THEN
	axis.cplOn(RatioNumerator := axis.setGearRatio.ratioNumeratorOut,
			Execute := axis.setGearRatio.trigger ,RatioDenominator := axis.setGearRatio.ratioDenominator,
			Acceleration := 40000, Deceleration := 40000);
	END_IF
	CASE StateCtrl OF
	CTRL_FIRST_START:
		busy := TRUE;
		StateCtrl := CTRL_EMERGENCYSTOP_BEFORE;

	CTRL_MANUAL_BEFORE:
		IF BetrCtrl.value = CONST.MACHINEMODES.MANUAL THEN
		(*	clamp.init(clk := clk);*)
			BetrStatus(set := TRUE, value := CONST.MACHINEMODES.MANUAL);
			chkStatus.enable := TRUE;
			err(reset := TRUE);
			busy := FALSE;
			timer(IN:= FALSE);
			state := ST_IDLE;
			(*manualFirst := TRUE;*)
			axis.ctrl.BasicControl.Parameter.Deceleration	:= 100000.0;
			axis.ctrl.BasicControl.Parameter.Acceleration	:= 100000.0;
//			axis.setGearRatio.init := TRUE; // OKrebs 09.12.15
			StateCtrl := CTRL_MANUAL;
		ELSIF BetrCtrl.value = CONST.MACHINEMODES.EMERGENCYSTOP THEN
			StateCtrl := CTRL_EMERGENCYSTOP_BEFORE;
		ELSIF BetrCtrl.value = CONST.MACHINEMODES.SAFETYSTOP THEN
			StateCtrl := CTRL_SAFETYSTOP_BEFORE;
		ELSIF BetrCtrl.value = CONST.MACHINEMODES.AUTOMATIC THEN
			StateCtrl := CTRL_AUTO_BEFORE;
		END_IF

	CTRL_MANUAL:
		IF BetrCtrl.value <> CONST.MACHINEMODES.MANUAL THEN
			err(reset := TRUE);
			busy := TRUE;
			StateCtrl := CTRL_MANUAL_AFTER;
//		ELSIF axis.ctrl.MC_ReadStatus_0.StandStill THEN
//			axis.ctrl.cmd := CONST.AXIS.START;
//				timer(IN := TRUE, PT := T#8s);
//				IF timer.Q THEN
		ELSE
				ac_manualConv;
		END_IF
		(*ELSE
			StateCtrl := CTRL_RESET_START;*)
		(*END_IF*)

	CTRL_MANUAL_AFTER:
		timer(IN:= FALSE);
		chkStatus.enable := FALSE;
		axis.ctrl.cmd := CONST.AXIS.NOACTION;
		ac_setStateAfterPB;

	CTRL_AUTO_BEFORE:
		IF BetrCtrl.value = CONST.MACHINEMODES.AUTOMATIC THEN
		BetrStatus(set := TRUE, value := CONST.MACHINEMODES.AUTOMATIC);
			(*clamp.init(clk := clk);*)
			err(reset := TRUE);
			chkStatus.enable := TRUE;
			busy := FALSE;
			state := ST_IDLE;
			axis.ctrl.BasicControl.Parameter.Deceleration	:= 100000.0;
			axis.ctrl.BasicControl.Parameter.Acceleration	:= 100000.0;
			StateCtrl := CTRL_AUTO;
		ELSIF BetrCtrl.value = CONST.MACHINEMODES.EMERGENCYSTOP THEN
			StateCtrl := CTRL_EMERGENCYSTOP_BEFORE;
		ELSIF BetrCtrl.value = CONST.MACHINEMODES.SAFETYSTOP THEN
			StateCtrl := CTRL_SAFETYSTOP_BEFORE;
		ELSIF BetrCtrl.value = CONST.MACHINEMODES.MANUAL THEN
			StateCtrl := CTRL_MANUAL_BEFORE;
		END_IF

	(* ******************************** *)
	(* *********** AUTO *************** *)
	(* ******************************** *)
	CTRL_AUTO:
		IF BetrCtrl.value <> CONST.MACHINEMODES.AUTOMATIC THEN
			err(reset := TRUE);
			busy := TRUE;
			StateCtrl := CTRL_AUTO_AFTER;
		ELSE
			;(*ac_automatic();*)
		END_IF

	CTRL_AUTO_AFTER:
		chkStatus.enable := FALSE;
		state := ST_IDLE;
		ac_setStateAfterPB;

	CTRL_STOP_BEFORE:
		IF BetrCtrl.value = CONST.MACHINEMODES.EMERGENCYSTOP THEN
			StateCtrl := CTRL_EMERGENCYSTOP_BEFORE;
		ELSIF BetrCtrl.value = CONST.MACHINEMODES.SAFETYSTOP THEN
			StateCtrl := CTRL_SAFETYSTOP_BEFORE;
		ELSE
			state := ST_IDLE;
			StateCtrl := CTRL_STOP;
		END_IF

	CTRL_STOP:
		IF BetrCtrl.value = CONST.MACHINEMODES.EMERGENCYSTOP THEN
			StateCtrl := CTRL_EMERGENCYSTOP_BEFORE;
		ELSIF BetrCtrl.value = CONST.MACHINEMODES.SAFETYSTOP THEN
			StateCtrl := CTRL_SAFETYSTOP_BEFORE;
		ELSE
			CASE state OF
			ST_IDLE:
				state := ST_QUIT;

			ST_QUIT:
				state := ST_IDLE;
				StateCtrl := CTRL_STOP_AFTER;
			END_CASE
		END_IF

	CTRL_STOP_AFTER:
		IF BetrCtrl.value = CONST.MACHINEMODES.EMERGENCYSTOP THEN
			StateCtrl := CTRL_EMERGENCYSTOP_BEFORE;
		ELSIF BetrCtrl.value = CONST.MACHINEMODES.SAFETYSTOP THEN
			StateCtrl := CTRL_SAFETYSTOP_BEFORE;
		ELSIF BetrCtrl.value = CONST.MACHINEMODES.MANUAL THEN
			StateCtrl := CTRL_MANUAL_BEFORE;
		ELSIF BetrCtrl.value = CONST.MACHINEMODES.AUTOMATIC THEN
			StateCtrl := CTRL_AUTO_BEFORE;
		END_IF

	CTRL_RESET_START:
		BetrStatus(set := TRUE,value := CONST.MACHINEMODES.RESET);
		IF BetrCtrl.value = CONST.MACHINEMODES.EMERGENCYSTOP THEN
			StateCtrl := CTRL_EMERGENCYSTOP_BEFORE;
		ELSIF BetrCtrl.value = CONST.MACHINEMODES.SAFETYSTOP THEN
			StateCtrl := CTRL_SAFETYSTOP_BEFORE;
		ELSE
			IF axis.ctrl.busy OR axis.ctrl.cmd <> CONST.AXIS.NOACTION  THEN
				axis.ctrl(cmd := CONST.AXIS.NOACTION);
//			ELSIF axis.ctrl.MC_ReadStatus_0.Disabled THEN
//				axis.ctrl(cmd := CONST.AXIS.RESET);
//				StateCtrl := CTRL_RESET;
			ELSE
				axis.ctrl(cmd := CONST.AXIS.RESET);
				StateCtrl := CTRL_RESET;
			END_IF
		END_IF

	CTRL_RESET:
		axis.ctrl();
		IF BetrCtrl.value = CONST.MACHINEMODES.EMERGENCYSTOP THEN
			StateCtrl := CTRL_EMERGENCYSTOP_BEFORE;
		ELSIF BetrCtrl.value = CONST.MACHINEMODES.SAFETYSTOP THEN
			StateCtrl := CTRL_SAFETYSTOP_BEFORE;
		ELSE
//			IF NOT axis.ctrl.busy THEN (* auskommentiert am 26.06..14*)
//				axis.ctrl(cmd := CONST.AXIS.NOACTION);
//				StateCtrl := CTRL_RESET_AFTER;
//			END_IF
			axis.ctrl(cmd := CONST.AXIS.POWER_OFF);
			StateCtrl := CTRL_RESET_AFTER;
		END_IF

	CTRL_RESET_AFTER:
		IF BetrCtrl.value = CONST.MACHINEMODES.RESET THEN
			busy := FALSE;
		ELSE
			busy := TRUE;
		(*	clamp.init(clk := clk);*)
			err(reset := TRUE);
			manualFirst := TRUE;
			IF BetrCtrl.value = CONST.MACHINEMODES.EMERGENCYSTOP THEN
				StateCtrl := CTRL_EMERGENCYSTOP_BEFORE;
			ELSIF BetrCtrl.value = CONST.MACHINEMODES.SAFETYSTOP THEN
				StateCtrl := CTRL_SAFETYSTOP_BEFORE;
			ELSIF BetrCtrl.value = CONST.MACHINEMODES.SAFETYSTOP THEN
				StateCtrl := CTRL_SAFETYSTOP_BEFORE;
			ELSIF BetrCtrl.value = CONST.MACHINEMODES.MANUAL  AND safety.valid THEN
				supplydelay(IN:= TRUE, PT := T#8s);
				IF supplydelay.Q THEN
					axis.ctrl(cmd := CONST.AXIS.POWER_ON);
					busy := TRUE;
					supplydelay(IN:= FALSE);
					StateCtrl := CTRL_MANUAL_BEFORE;
				END_IF
			ELSIF BetrCtrl.value = CONST.MACHINEMODES.AUTOMATIC  AND safety.valid THEN
				supplydelay(IN:= TRUE, PT := T#8s);
				IF supplydelay.Q THEN
					axis.ctrl(cmd := CONST.AXIS.POWER_ON);
					busy := TRUE;
					supplydelay(IN:= FALSE);
					StateCtrl := CTRL_AUTO_BEFORE;
				END_IF
			END_IF
		END_IF

	CTRL_SAFETYSTOP_BEFORE:
		status.isCoupled := FALSE;
		status.ready := FALSE;
//		IF BetrCtrl.value = CONST.MACHINEMODES.EMERGENCYSTOP THEN
//			StateCtrl := CTRL_EMERGENCYSTOP_BEFORE;
//		ELSE
//			BetrStatus(set := TRUE,value := CONST.MACHINEMODES.SAFETYSTOP);
//			state := ST_IDLE;
//			axis.ctrl.verzoegerung	:= 1600000.0;
//			axis.ctrl(cmd := CONST.AXIS.STOP);
//			StateCtrl := CTRL_SAFETYSTOP;
			//		END_IF	status.isCoupled := FALSE;
		//12.03.15
		IF BetrCtrl.value = CONST.MACHINEMODES.EMERGENCYSTOP THEN
				StateCtrl := CTRL_EMERGENCYSTOP_BEFORE;
		ELSE
			BetrStatus(set := TRUE,value := CONST.MACHINEMODES.SAFETYSTOP);
			state := ST_IDLE;
			manualFirst := FALSE;
			axis.ctrl.verzoegerung	:= CONST.AXIS.EMERGENCY_DECELERATION;
			axis.ctrl.cmd := CONST.AXIS.STOP;
			StateCtrl := CTRL_SAFETYSTOP;
		END_IF

		CTRL_SAFETYSTOP:

		IF BetrCtrl.value = CONST.MACHINEMODES.EMERGENCYSTOP THEN
			StateCtrl := CTRL_EMERGENCYSTOP_BEFORE;
		ELSE
			BetrStatus(set := TRUE,value := CONST.MACHINEMODES.SAFETYSTOP);
			IF axis.ctrl.MC_ReadStatus_0.StandStill THEN
				axis.ctrl.cmd := CONST.AXIS.POWER_OFF;
			ELSIF axis.ctrl.MC_ReadStatus_0.Disabled THEN
				axis.ctrl.cmd := CONST.AXIS.NOACTION;
				StateCtrl := CTRL_SAFETYSTOP_AFTER;
			END_IF
		END_IF

	CTRL_SAFETYSTOP_AFTER:
		busy := FALSE;
		manualFirst := TRUE;
		status.ready := FALSE;
		IF BetrCtrl.value = CONST.MACHINEMODES.EMERGENCYSTOP THEN
			busy := TRUE;
			StateCtrl := CTRL_EMERGENCYSTOP_BEFORE;
		ELSIF BetrCtrl.value = CONST.MACHINEMODES.MANUAL  AND safety.valid THEN
				IF axis.ctrl.MC_ReadStatus_0.Errorstop THEN
					axis.ctrl(cmd := CONST.AXIS.RESET);
				END_IF
				supplydelay(IN:= TRUE, PT := T#8s);
				IF supplydelay.Q THEN
					axis.ctrl(cmd := CONST.AXIS.POWER_ON);
					(*axis.ctrl(cmd := CONST.AXIS.NOACTION);*)
					busy := TRUE;
					supplydelay(IN:= FALSE);
					StateCtrl := CTRL_MANUAL_BEFORE;
				END_IF
		ELSIF BetrCtrl.value = CONST.MACHINEMODES.AUTOMATIC  AND safety.valid THEN
				IF axis.ctrl.MC_ReadStatus_0.Errorstop THEN
					axis.ctrl(cmd := CONST.AXIS.RESET);
				END_IF
				supplydelay(IN:= TRUE, PT := T#8s);
				IF supplydelay.Q THEN
					axis.ctrl(cmd := CONST.AXIS.POWER_ON);
				(*	axis.ctrl(cmd := CONST.AXIS.NOACTION);*)
					busy := TRUE;
					supplydelay(IN:= FALSE);
					StateCtrl := CTRL_AUTO_BEFORE;
				END_IF
		END_IF

	CTRL_EMERGENCYSTOP_BEFORE:
//		status.isCoupled := FALSE;
//		status.ready := FALSE;
//		axis.ctrl(cmd := CONST.AXIS.POWER_OFF);
//		BetrStatus(set := TRUE, value := CONST.MACHINEMODES.EMERGENCYSTOP);
//		busy := FALSE;
//		StateCtrl := CTRL_EMERGENCYSTOP;
		status.isCoupled := FALSE;
		status.ready := FALSE;
		manualFirst := TRUE;
		BetrStatus(set := TRUE, value := CONST.MACHINEMODES.EMERGENCYSTOP);
		IF  axis.ctrl.MC_ReadStatus_0.ContinuousMotion OR axis.ctrl.MC_ReadStatus_0.DiscreteMotion
			OR axis.ctrl.MC_ReadStatus_0.SynchronizedMotion THEN //alle Zustände in denen die Achse sich bewegen kann
			axis.ctrl.verzoegerung:= CONST.AXIS.EMERGENCY_DECELERATION; (*200m/min in 3 sek*); (* von 200m/min in 2 sek*)
			axis.ctrl.cmd := CONST.AXIS.STOP;
			state := ST_IDLE;
			StateCtrl := CTRL_EMERGENCYSTOP;
		ELSE //wenn die Maschine eingeschaltet wird
			axis.ctrl.cmd := CONST.AXIS.NOACTION;
			state := ST_IDLE;
			StateCtrl := CTRL_EMERGENCYSTOP;
		END_IF

	CTRL_EMERGENCYSTOP:
		status.isCoupled := FALSE;
		status.ready := FALSE;
		IF BetrCtrl.value = CONST.MACHINEMODES.EMERGENCYSTOP THEN
			IF axis.ctrl.MC_ReadStatus_0.StandStill THEN
				axis.ctrl.cmd := CONST.AXIS.POWER_OFF;
				busy := FALSE;
			ELSIF axis.ctrl.MC_ReadStatus_0.Disabled THEN
				axis.ctrl.cmd := CONST.AXIS.NOACTION;
				busy := FALSE;
			END_IF
		ELSE
			busy := TRUE;
			timer(IN := TRUE, PT := T#2s);
			StateCtrl := CTRL_EMERGENCYSTOP_AFTER;
		END_IF

	CTRL_EMERGENCYSTOP_AFTER:
		timer();
		IF BetrCtrl.value = CONST.MACHINEMODES.EMERGENCYSTOP THEN
			timer(IN := FALSE);
			BetrStatus(set := TRUE , value := CONST.MACHINEMODES.EMERGENCYSTOP);
			busy := FALSE;
			StateCtrl := CTRL_EMERGENCYSTOP;
		ELSIF timer.Q THEN
			timer(IN := FALSE);
			StateCtrl := CTRL_RESET_START;
		END_IF

	ELSE
		;
	END_CASE

END_FUNCTION_BLOCK
```

#### FB_ConveyorConfig.st
```iecst
(********************************************************************
 * COPYRIGHT -- Microsoft
 ********************************************************************
 * Programm: MAIN
 * Datei: FB_ConveyorConfig.st
 * Autor: Awalz
 * Erstellt: 12. Mai 2014
 ********************************************************************
 * Implementierung des Programms MAIN
 ********************************************************************)

 (*<$Description$> TODO: Bitte Kommentar hier einzufügen </$Description$>*)
FUNCTION_BLOCK FB_ConveyorConfig
	TOF_delay.PT := T#1s;  //OKrebs 08.09.21
	TOF_delay.PT := T#1s;  //OKrebs 08.09.21
	axis.cplOn( Master := machineMasterCtrl.AxisREF, Slave := axis.ctrl.AxisREF);
 	axis.cplOff( Slave := axis.ctrl.AxisREF);
	CASE state OF
	ST_IDLE:
		IF cmd <> CONST.CUTTINGUNIT.CMDs.NO_CMD THEN
			busy := TRUE;
			err(reset:= TRUE);
			cmdtmp := cmd;
			IF cmd = CONST.CUTTINGUNIT.CMDs.CPL_ON THEN
				state := ST_CPL_START;
			ELSIF cmd = CONST.CUTTINGUNIT.CMDs.CPL_OFF THEN
				state := ST_CPLOFF_START;
			ELSIF  cmd =  CONST.CUTTINGUNIT.CMDs.MOVEBW OR cmd = CONST.CUTTINGUNIT.CMDs.MOVEFW THEN
				state := ST_MOVE_START;
			ELSE
				err.state := state;
				err(text := 'CommandError');
				state := ST_ERROR;
			END_IF
		END_IF

	ST_CPL_START:
		axis.ctrl();

		IF cmd = CONST.CUTTINGUNIT.CMDs.ABORT THEN
			state := ST_ABORT;
		ELSIF axis.cplOn.InGear THEN
			status.isCoupled := TRUE;
			status.mode := CONST.UNITMODEs.ENABLE;
			state := ST_QUIT;
		ELSIF axis.cplOn.Busy  THEN
			status.isCoupled := TRUE;
			status.mode := CONST.UNITMODEs.ENABLE;
			state := ST_QUIT;
		ELSIF axis.ctrl.MC_ReadStatus_0.StandStill THEN
			axis.cplOn(Execute := TRUE, Master := machineMasterCtrl.AxisREF, Slave := axis.ctrl.AxisREF,
			Acceleration := 20000, Deceleration := 20000 , RatioDenominator := 1000, RatioNumerator := axis.setGearRatio.ratioDenominator(* 1000*));
			state := ST_CPL_WAIT;
		END_IF

	ST_CPL_WAIT:
		axis.cplOn( Master := machineMasterCtrl.AxisREF, Slave := axis.ctrl.AxisREF );
		IF axis.cplOn.Busy THEN
			axis.cplOn(Execute := FALSE, Master := machineMasterCtrl.AxisREF, Slave := axis.ctrl.AxisREF);
				status.isCoupled := TRUE;
				status.mode := CONST.UNITMODEs.ENABLE;
				state := ST_QUIT;
		ELSIF axis.cplOn.Error THEN
				err.id := axis.cplOn.ErrorID;
				err.fnc := 'axis.cplOn';
				err.state := state;
				state := ST_ERROR;
(*			ELSIF axis.cplOn.CommandAborted THEN
				err.fnc := 'axis.cplOn CommandAborted';
				err.state := state;
				state := ST_ERROR;
			ELSIF axis.cplOn.InGear THEN *)
		END_IF

	ST_CPLOFF_START:
		IF cmd = CONST.CUTTINGUNIT.CMDs.ABORT THEN
			state := ST_ABORT;
		ELSIF axis.cplOff.Error  THEN
			err.state := state;
			err.text := 'MC_GearOut';
			state := ST_ERROR;
		ELSIF axis.cplOff.Busy OR axis.cplOff.Execute THEN
			axis.cplOff(Execute := FALSE, Slave := axis.ctrl.AxisREF );
		ELSE
			axis.cplOff(Execute := TRUE, Slave := axis.ctrl.AxisREF);
			state := ST_CPLOFF_WAIT;
		END_IF

	ST_CPLOFF_WAIT:
		axis.cplOff( Slave := axis.ctrl.AxisREF );
		IF  axis.cplOff.Done THEN
			IF axis.cplOff.Error THEN
				err.id := axis.cplOff.ErrorID;
				err.fnc := 'axis.cplOff';
				err.state := state;
				state := ST_ERROR;
			ELSE
				axis.cplOff.Execute := FALSE;
				status.isCoupled := FALSE;
				IF cmd = CONST.CUTTINGUNIT.CMDs.MOVEBW OR cmd = CONST.CUTTINGUNIT.CMDs.MOVEFW THEN
					state := ST_MOVE_START;
				ELSE

					state := ST_QUIT;
				END_IF
			END_IF

		END_IF
//	ST_MOVE_START:
//			//		masterAxis.ctrl.ref.ReadStatus();
//		IF cmd = CONST.CUTTINGUNIT.CMDs.NO_CMD THEN
//			busy := FALSE;
//			state := ST_IDLE;
//		ELSIF axis.ctrl.MC_ReadStatus_0.SynchronizedMotion THEN
//				//			err.text := 'MOVE nicht möglich. Achse ist gekoppelt';
//				//			err.state := state;
//			state := ST_CPLOFF_START;
//				//		ELSIF status.isCalibrated THEN (* die Stanze soll man auch ohne zu rferenzieren drehen können*)
//				//			IF axis.ctrl.busy (*OR axis.ctrl.cmd <> CONST.AXIS.NOACTION*) THEN
//				//				axis.ctrl(cmd := CONST.AXIS.NOACTION);
//		ELSIF axis.ctrl.MC_ReadStatus_0.StandStill OR axis.ctrl.MC_ReadStatus_0.ContinuousMotion THEN
//			IF cmd = CONST.CUTTINGUNIT.CMDs.MOVEBW THEN
//				axis.ctrl(cmd := CONST.AXIS.JOG_NEG, velocity := 4);
//				state := ST_MOVE_WAIT;
//			ELSE
//				axis.ctrl(cmd := CONST.AXIS.JOG_POS, velocity := 4);
//				state := ST_MOVE_WAIT;
//			END_IF
//		END_IF

		//***********************neu********************// OKrebs 14.01.16
		ST_MOVE_START:// 40
			TON_delay.IN := cmd = CONST.CUTTINGUNIT.CMDs.MOVEBW OR cmd = CONST.CUTTINGUNIT.CMDs.MOVEFW;  //OKrebs 08.09.21
			TOF_delay.IN := cmd = CONST.CUTTINGUNIT.CMDs.MOVEBW OR cmd = CONST.CUTTINGUNIT.CMDs.MOVEFW;  //OKrebs 08.09.21
			IF NOT axis.MC_BR_Phasing_0.Busy  AND axis.ctrl.MC_ReadStatus_0.SynchronizedMotion AND cmd <> CONST.CUTTINGUNIT.CMDs.NO_CMD THEN
				IF cmd = CONST.CUTTINGUNIT.CMDs.MOVEBW AND TON_delay.Q THEN
					axis.MC_BR_Phasing_0.Acceleration := 90000;
					axis.MC_BR_Phasing_0.ApplicationMode := mcVELOCITY_CONTROL ;
					axis.MC_BR_Phasing_0.Slave := axis.ctrl.AxisREF;
					axis.MC_BR_Phasing_0.Velocity := - 16666.67 * 3; //1m/min
					axis.MC_BR_Phasing_0.Enable := TRUE;
					axis.MC_BR_Phasing_0.InitData := TRUE;
					axis.MC_BR_Phasing_0.PerformVelocityControl := TRUE;
				ELSIF cmd = CONST.CUTTINGUNIT.CMDs.MOVEFW AND TON_delay.Q THEN
					axis.MC_BR_Phasing_0.Acceleration := 90000;
					axis.MC_BR_Phasing_0.ApplicationMode := mcVELOCITY_CONTROL;
					axis.MC_BR_Phasing_0.Slave := axis.ctrl.AxisREF;
					axis.MC_BR_Phasing_0.Velocity := 16666.67 * 3; //1m/min
					axis.MC_BR_Phasing_0.Enable := TRUE;
					axis.MC_BR_Phasing_0.InitData := TRUE;
					axis.MC_BR_Phasing_0.PerformVelocityControl := TRUE;
				END_IF
			ELSIF cmd =  CONST.CUTTINGUNIT.CMDs.NO_CMD AND axis.ctrl.MC_ReadStatus_0.SynchronizedMotion THEN
				axis.MC_BR_Phasing_0.Velocity := 0;
				axis.MC_BR_Phasing_0.PerformVelocityControl := FALSE;
				axis.MC_BR_Phasing_0.InitData := FALSE;
				IF axis.MC_BR_Phasing_0.ShiftAttained OR EDGENEG(TOF_delay.Q) THEN
					axis.MC_BR_Phasing_0.Enable := FALSE;
					state := ST_QUIT;
				END_IF
			ELSIF cmd =  CONST.CUTTINGUNIT.CMDs.NO_CMD AND (axis.ctrl.MC_ReadStatus_0.StandStill OR axis.ctrl.MC_ReadStatus_0.ContinuousMotion) THEN
				axis.ctrl(cmd := CONST.AXIS.NOACTION);
				state := ST_QUIT;
			ELSIF  axis.ctrl.MC_ReadStatus_0.Disabled THEN
				state := ST_QUIT;
			ELSE

			END_IF

		//******************************************************************************

	ST_MOVE_WAIT:
		axis.ctrl();
		IF cmd = CONST.CUTTINGUNIT.CMDs.NO_CMD THEN
			axis.ctrl(cmd := CONST.AXIS.NOACTION );
			state := ST_MOVE_QUIT;
		END_IF
		//
	ST_MOVE_QUIT: (* hier evtl. koppeln*)
		state := ST_CPL_START;
		(*state := ST_QUIT;*)
	ST_ERROR:
		IF LEN(err.fnc) < 1 THEN
			err.fnc := 'FB_ConveyorConfig';
		END_IF
		err.flag := TRUE;
		state := ST_QUIT;

	ST_ABORT:
		state := ST_ABORT_QUIT;

	ST_ABORT_QUIT:
		busy := FALSE;
		IF cmd <> CONST.CUTTINGUNIT.CMDs.NO_CMD THEN
			state := ST_IDLE;
		END_IF

	ST_QUIT:
		IF cmd = CONST.CUTTINGUNIT.CMDs.ABORT THEN
			busy := TRUE;
			state := ST_ABORT;
		ELSE
			busy := FALSE;
			IF cmd = CONST.CUTTINGUNIT.CMDs.NO_CMD THEN
				state := ST_IDLE;
			END_IF
		END_IF
	END_CASE
	axis.MC_BR_Phasing_0();	//OKrebs 14.01.16
	TOF_delay(); //OKrebs 08.09.21
	TON_delay(); //OKrebs 08.09.21
END_FUNCTION_BLOCK
```

#### FB_CONVEYOR.st
```iecst
(********************************************************************
 * COPYRIGHT -- Microsoft
 ********************************************************************
 * Programm: MAIN
 * Datei: FB_CONVEYOR.st
 * Autor: Awalz
 * Erstellt: 12. Mai 2014
 ********************************************************************
 * Implementierung des Programms MAIN
 ********************************************************************)

 (*<$Description$> TODO: Bitte Kommentar hier einzufügen </$Description$>*)
FUNCTION_BLOCK FB_CONVEYOR
END_FUNCTION_BLOCK
```

#### Package Logical/MainMachineCtrl/MAIN/General - Neues leeres Paket

#### FB_GlobalMachineVar.st
```iecst
(********************************************************************
 * COPYRIGHT -- Microsoft
 ********************************************************************
 * Programm: MAIN
 * Datei: FB_GlobalMachineVar.st
 * Autor: Awalz
 * Erstellt: 5. Juni 2014
 ********************************************************************
 * Implementierung des Programms MAIN
 ********************************************************************)

 (*<$Description$> TODO: Bitte Kommentar hier einzufügen </$Description$>*)
FUNCTION_BLOCK FB_GlobalMachineVar
END_FUNCTION_BLOCK
```

#### Package Logical/MainMachineCtrl/MAIN/Stati_Message - Neues leeres Paket

#### FB_UnitsStatus.st
```iecst
(********************************************************************
 * COPYRIGHT -- Microsoft
 ********************************************************************
 * Programm: MAIN
 * Datei: FB_UnitsStatus.st
 * Autor: Awalz
 * Erstellt: 1. April 2014
 ********************************************************************
 * Implementierung des Programms MAIN
 ********************************************************************)

 (*<$Description$> TODO: Bitte Kommentar hier einzufügen </$Description$>*)
FUNCTION_BLOCK FB_UnitsStatus
//	pullbreak();21.09.15
//	pullbreakSt();
//	longcutter();
//	conveyor();
//	catchbelt();
//	UnwinderUnit();
	ready := (longcutter.axis.ctrl.MC_ReadStatus_0.SynchronizedMotion AND pullbreak.status.ready AND pullbreakSt.status.ready AND pullbreakSt.hubctrl.isdown AND conveyor.status.ready AND catchbelt.status.ready AND cuttingunit1.status.isCalibrated AND cuttingunit2.status.isCalibrated AND webbuffer.axis.ctrl.BasicControl.AxisState.Homed AND turngridwinder.feeder.BasicControl.AxisState.Homed); // OKrebs 09.12.15
	diameterStop:= UnwinderUnit.unwinderDrv.ctrl.diameterStop OR UnwinderUnit.unwinderOp.ctrl.diameterStop;
	diameterwarning:= UnwinderUnit.unwinderDrv.ctrl.diameterWarning OR UnwinderUnit.unwinderOp.ctrl.diameterWarning;
	clampingfront:=  UnwinderUnit.clamp.toDown_o OR UnwinderUnit.unwinderDrv.clamp.toDown_o OR UnwinderUnit.unwinderOp.clamp.toDown_o;
	clampingsplicetable := UnwinderUnit.splicetable.clampAfter.toDown_o OR UnwinderUnit.splicetable.clampBefore.toDown_o;
	clampingback:= longcutter.webclamp.toDown_o;

END_FUNCTION_BLOCK
```

#### Package Logical/MainMachineCtrl/MAIN/Winder - Neues leeres Paket

#### FB_WinderCtrl.st
```iecst
(********************************************************************
 * COPYRIGHT -- Microsoft
 ********************************************************************
 * Programm: MAIN
 * Datei: FB_WinderCtrl.st
 * Autor: okrebs
 * Erstellt: 6. Mai 2014
 ********************************************************************
 * Implementierung des Programms MAIN
 ********************************************************************)

(* TODO: Bitte Kommentar hier einzufügen *)
FUNCTION_BLOCK FB_WinderCtrl
	winderaxis(machineaxis := machineMaster, data := data, (*status := status*));
	(*die Daten später von der Visu bzw. dem Rezept setzen*)
	data.machData.frictionCompensation := 3;
	data.recipeData.minDiamTension := 20;
	data.recipeData.maxDiamTension := 80;
	(* und auch auf Kraft N normieren *)
//	data.recipeData.mode := CONST.UNITMODEs.ENABLE;

//status.modeName := CONST.UNITMODEs.texts[1];
	status.ready := (*winderaxis.MC_ReadStatus_0.ContinuousMotion OR (AND *) NOT winderaxis.MC_ReadStatus_0.Disabled AND NOT winderaxis.MC_TorqueControl_0.Error;
	CASE StateCtrl OF
		CTRL_FIRST_START:
			busy := TRUE;
			StateCtrl := CTRL_EMERGENCYSTOP_BEFORE;
		CTRL_MANUAL_BEFORE:
			IF BetrCtrl.value = CONST.MACHINEMODES.MANUAL THEN
				BetrStatus(set := TRUE,value := CONST.MACHINEMODES.MANUAL);
				busy := FALSE;
				(*clamp.init(clk := clk);*)
				chkStatus.enable := TRUE;
				err(reset := TRUE);
				timer(IN:= FALSE);
				state := ST_IDLE;
				firstStart := TRUE;
				StateCtrl := CTRL_MANUAL;
			ELSIF BetrCtrl.value = CONST.MACHINEMODES.EMERGENCYSTOP THEN
				StateCtrl := CTRL_EMERGENCYSTOP_BEFORE;
			ELSIF BetrCtrl.value = CONST.MACHINEMODES.SAFETYSTOP THEN
				StateCtrl := CTRL_SAFETYSTOP_BEFORE;
			ELSIF BetrCtrl.value = CONST.MACHINEMODES.AUTOMATIC THEN
				StateCtrl := CTRL_AUTO_BEFORE;
			END_IF

		CTRL_MANUAL:
			IF BetrCtrl.value <> CONST.MACHINEMODES.MANUAL THEN
				err(reset := TRUE);
				busy := TRUE;
				StateCtrl := CTRL_MANUAL_AFTER;
			ELSE
				(*winderaxis.enable := TRUE;*)
				ac_manualWinder; (*Aufruf der Action*)
			END_IF

		CTRL_MANUAL_AFTER:
			chkStatus.enable := FALSE;
		ac_setStateAfterWinder; (*Aufruf der Action*)

		CTRL_AUTO_BEFORE:
			IF BetrCtrl.value = CONST.MACHINEMODES.AUTOMATIC THEN
				BetrStatus(set := TRUE, value := CONST.MACHINEMODES.AUTOMATIC);
			(*clamp.init(clk := clk);*)
			chkStatus.enable := TRUE;
				err(reset := TRUE);
				busy := FALSE;
				state := ST_IDLE;
				winderaxis.enable := TRUE;
				StateCtrl := CTRL_AUTO;
			ELSIF BetrCtrl.value = CONST.MACHINEMODES.EMERGENCYSTOP THEN
				StateCtrl := CTRL_EMERGENCYSTOP_BEFORE;
			ELSIF BetrCtrl.value = CONST.MACHINEMODES.SAFETYSTOP THEN
				StateCtrl := CTRL_SAFETYSTOP_BEFORE;
			ELSIF BetrCtrl.value = CONST.MACHINEMODES.MANUAL THEN
				StateCtrl := CTRL_MANUAL_BEFORE;
			END_IF

		(* ******************************** *)
		(* *********** AUTO *************** *)
		(* ******************************** *)
		CTRL_AUTO:
			IF BetrCtrl.value <> CONST.MACHINEMODES.AUTOMATIC THEN
				err(reset := TRUE);
				busy := TRUE;
				StateCtrl := CTRL_AUTO_AFTER;
			ELSE
				winderaxis.cmd := CONST.AXIS.START;
				(*ac_automatic();*)
			END_IF

		CTRL_AUTO_AFTER:
			chkStatus.enable := FALSE;
			winderaxis.cmd := CONST.AXIS.STOP;
			state := ST_IDLE;
			ac_setStateAfterWinder;

		CTRL_STOP_BEFORE:
			IF BetrCtrl.value = CONST.MACHINEMODES.EMERGENCYSTOP THEN
				StateCtrl := CTRL_EMERGENCYSTOP_BEFORE;
			ELSIF BetrCtrl.value = CONST.MACHINEMODES.SAFETYSTOP THEN
				StateCtrl := CTRL_SAFETYSTOP_BEFORE;
			ELSE
				state := ST_IDLE;
				StateCtrl := CTRL_STOP;
			END_IF

		CTRL_STOP:
			IF BetrCtrl.value = CONST.MACHINEMODES.EMERGENCYSTOP THEN
				StateCtrl := CTRL_EMERGENCYSTOP_BEFORE;
			ELSIF BetrCtrl.value = CONST.MACHINEMODES.SAFETYSTOP THEN
				StateCtrl := CTRL_SAFETYSTOP_BEFORE;
			ELSE
				CASE state OF
					ST_IDLE:
						state := ST_QUIT;

					ST_QUIT:
						state := ST_IDLE;
						StateCtrl := CTRL_STOP_AFTER;
				END_CASE
			END_IF

		CTRL_STOP_AFTER:
			IF BetrCtrl.value = CONST.MACHINEMODES.EMERGENCYSTOP THEN
				StateCtrl := CTRL_EMERGENCYSTOP_BEFORE;
			ELSIF BetrCtrl.value = CONST.MACHINEMODES.SAFETYSTOP THEN
				StateCtrl := CTRL_SAFETYSTOP_BEFORE;
			ELSIF BetrCtrl.value = CONST.MACHINEMODES.MANUAL THEN
				StateCtrl := CTRL_MANUAL_BEFORE;
			ELSIF BetrCtrl.value = CONST.MACHINEMODES.AUTOMATIC THEN
				StateCtrl := CTRL_AUTO_BEFORE;
			END_IF

		CTRL_RESET_START:
			BetrStatus.set := TRUE;
			BetrStatus.value := CONST.MACHINEMODES.RESET;
			IF BetrCtrl.value = CONST.MACHINEMODES.EMERGENCYSTOP THEN
				StateCtrl := CTRL_EMERGENCYSTOP_BEFORE;
			ELSIF BetrCtrl.value = CONST.MACHINEMODES.SAFETYSTOP THEN
				StateCtrl := CTRL_SAFETYSTOP_BEFORE;
			ELSE
				IF winderaxis.busy  OR winderaxis.cmd <> CONST.AXIS.NOACTION THEN
					winderaxis(cmd := CONST.AXIS.NOACTION, machineaxis := machineMaster, data := data(*, status := status*));
				ELSE
					winderaxis(cmd := CONST.AXIS.RESET, machineaxis := machineMaster, data := data(*, status := status*));
					StateCtrl := CTRL_RESET;
				END_IF
			END_IF

		CTRL_RESET:
			winderaxis(machineaxis := machineMaster, data := data(*, status := status*));
			IF BetrCtrl.value = CONST.MACHINEMODES.EMERGENCYSTOP THEN
				StateCtrl := CTRL_EMERGENCYSTOP_BEFORE;
			ELSIF BetrCtrl.value = CONST.MACHINEMODES.SAFETYSTOP THEN
				StateCtrl := CTRL_SAFETYSTOP_BEFORE;
			ELSE
				IF NOT winderaxis.busy THEN
					winderaxis.cmd := CONST.AXIS.NOACTION;
					StateCtrl := CTRL_RESET_AFTER;
				END_IF
			END_IF

		CTRL_RESET_AFTER:
			IF BetrCtrl.value = CONST.MACHINEMODES.RESET THEN
				busy := FALSE;
			ELSE
				busy := TRUE;
			(*clamp.init(clk := clk);*)
				err(reset := TRUE);
				IF BetrCtrl.value = CONST.MACHINEMODES.EMERGENCYSTOP THEN
					StateCtrl := CTRL_EMERGENCYSTOP_BEFORE;
				ELSIF BetrCtrl.value = CONST.MACHINEMODES.SAFETYSTOP THEN
					StateCtrl := CTRL_SAFETYSTOP_BEFORE;
				ELSIF BetrCtrl.value = CONST.MACHINEMODES.SAFETYSTOP THEN
					StateCtrl := CTRL_SAFETYSTOP_BEFORE;
				ELSIF BetrCtrl.value = CONST.MACHINEMODES.MANUAL THEN
					supplydelay(IN:= TRUE, PT := T#8s);
					IF supplydelay.Q THEN
						winderaxis.cmd := CONST.AXIS.POWER_ON;
						busy := TRUE;
						supplydelay(IN:= FALSE);
						StateCtrl := CTRL_MANUAL_BEFORE;
					END_IF
				ELSIF BetrCtrl.value = CONST.MACHINEMODES.AUTOMATIC THEN
					supplydelay(IN:= TRUE, PT := T#8s);
					IF supplydelay.Q THEN
						winderaxis.cmd := CONST.AXIS.POWER_ON;
						busy := TRUE;
						supplydelay(IN:= FALSE);
						StateCtrl := CTRL_AUTO_BEFORE;
					END_IF
				END_IF
			END_IF

		CTRL_SAFETYSTOP_BEFORE:
			IF BetrCtrl.value = CONST.MACHINEMODES.EMERGENCYSTOP THEN
				StateCtrl := CTRL_EMERGENCYSTOP_BEFORE;
			ELSE
				BetrStatus.set := TRUE;
				BetrStatus.value := CONST.MACHINEMODES.SAFETYSTOP;
				state := ST_IDLE;
				StateCtrl := CTRL_SAFETYSTOP;
			END_IF

		CTRL_SAFETYSTOP:
			IF BetrCtrl.value = CONST.MACHINEMODES.EMERGENCYSTOP THEN
				StateCtrl := CTRL_EMERGENCYSTOP_BEFORE;
			ELSE
				CASE state OF
					ST_IDLE:
						state := ST_QUIT;

					ST_QUIT:
						state := ST_QUIT;
						StateCtrl := CTRL_SAFETYSTOP_AFTER;
				END_CASE
			END_IF

		CTRL_SAFETYSTOP_AFTER:
			busy := FALSE;
			IF BetrCtrl.value = CONST.MACHINEMODES.EMERGENCYSTOP THEN
				busy := TRUE;
				StateCtrl := CTRL_EMERGENCYSTOP_BEFORE;
			ELSIF BetrCtrl.value = CONST.MACHINEMODES.MANUAL THEN
				supplydelay(IN:= TRUE, PT := T#8s);
				IF supplydelay.Q THEN
					winderaxis.cmd := CONST.AXIS.POWER_ON;;
					busy := TRUE;
					supplydelay(IN:= FALSE);
					StateCtrl := CTRL_MANUAL_BEFORE;
				END_IF
			ELSIF BetrCtrl.value = CONST.MACHINEMODES.AUTOMATIC THEN
					supplydelay(IN:= TRUE, PT := T#8s);
				IF supplydelay.Q THEN
					winderaxis.cmd := CONST.AXIS.POWER_ON;
					busy := TRUE;
					supplydelay(IN:= FALSE);
					StateCtrl := CTRL_AUTO_BEFORE;
				END_IF
			END_IF

		CTRL_EMERGENCYSTOP_BEFORE:
			(*axis.drvCtrl.resetRelease(ref := axis.ctrl.ref);*)
			BetrStatus(set := TRUE,value := CONST.MACHINEMODES.EMERGENCYSTOP);
			(*mode.status.set(value := CONST.MACHINEMODES.EMERGENCYSTOP);*)
			busy := FALSE;
			StateCtrl := CTRL_EMERGENCYSTOP;

		CTRL_EMERGENCYSTOP:
			winderaxis.cmd := CONST.AXIS.POWER_OFF;
			IF BetrCtrl.value = CONST.MACHINEMODES.EMERGENCYSTOP THEN
				;
			ELSE
				busy := TRUE;
				timer(IN := TRUE, PT := T#2s);
				StateCtrl := CTRL_EMERGENCYSTOP_AFTER;
			END_IF

		CTRL_EMERGENCYSTOP_AFTER:
			timer();
			IF BetrCtrl.value = CONST.MACHINEMODES.EMERGENCYSTOP THEN
				timer(IN := FALSE);
				BetrStatus(set := TRUE,value := CONST.MACHINEMODES.EMERGENCYSTOP);
				busy := FALSE;
				StateCtrl := CTRL_EMERGENCYSTOP;
			ELSIF timer.Q THEN
				timer(IN := FALSE);
				StateCtrl := CTRL_RESET_START;
			END_IF

		ELSE
			;
	END_CASE
END_FUNCTION_BLOCK
```

#### FB_Winder.st
```iecst
(********************************************************************
 * COPYRIGHT -- Microsoft
 ********************************************************************
 * Programm: MAIN
 * Datei: FB_TandemWinder.st
 * Autor: okrebs
 * Erstellt: 6. Mai 2014
 ********************************************************************
 * Implementierung des Programms MAIN
 ********************************************************************)

(* TODO: Bitte Kommentar hier einzufügen *)
FUNCTION_BLOCK FB_Winder
END_FUNCTION_BLOCK
```

#### FB_WinderAxis.st
```iecst
(********************************************************************
 * COPYRIGHT -- Microsoft
 ********************************************************************
 * Programm: MAIN
 * Datei: FB_Winder.st
 * Autor: okrebs
 * Erstellt: 6. Mai 2014
 ********************************************************************
 * Implementierung des Programms MAIN
 ********************************************************************)

(* TODO: Bitte Kommentar hier einzufügen *)
FUNCTION_BLOCK FB_WinderAxis
	IF firststart THEN
		//**********	diameter estimation	Top winder ****************
		// set winder parameters
		pAxis ACCESS AxisREF;
		pMasteraxisREF ACCESS machineaxis.AxisREF;
		SysPara.minDiam			:= 80; //gMachRecipe.Winders.CoreDiam; // [mm]
		SysPara.xDiam			:= 80; //gMachRecipe.Winders.CoreDiam; // [mm]
		SysPara.maxDiam			:= 600; //gMachRecipe.topTandemWind.StopDiam; // [mm]
		SysPara.minInertia		:= 1.0; // [kgm^2]
		SysPara.xInertia		:= 1.0; // [kgm^2]
		SysPara.gearRatio		:= data.machData.GEAR_RATIO; // [1]GEAR_RATIO_TOP_TWIND;
		SysPara.kvTorque		:= 0.01; // [Nms]
		SysPara.posTorque		:= 0.1; // [Nm]
		SysPara.negTorque		:= 0.1; // [Nm]
		SysPara.matThickness	:= 200.00; // [um]
		SysPara.wndWidth		:= 650.00; // [mm]
		SysPara.lineUnits		:= 1000000; // [units/m]
		SysPara.wndUnits		:= pAxis.encoder_if.parameter.scaling.load.units; // gTWindTop.encoder_if.parameter.scaling.load.units; 	// [units]
		SysPara.revMotor		:= pAxis.encoder_if.parameter.scaling.load.rev_motor; // gTWindTop.encoder_if.parameter.scaling.load.rev_motor; // [units]
		SysPara.axisType		:= data.machData.axistyp; (*-1;*) // rewinder (* (-1: winder, +1: unwinder).*)

		EstPara.cycEstTrig 		:= 100; // [units]
		EstPara.cycEstWindow 	:= 100; // [units]
		EstPara.filterMode 		:= 2; // LQ filter
		EstPara.filterWindow 	:= 300; // 3 times cycEstTrig

		WNCCalcDiam_0.pSysPara	:= ADR(SysPara);
		WNCCalcDiam_0.pEstPara	:= ADR(EstPara);
		//**************************************************
		firststart := FALSE;

	END_IF
	(********************MC_BR_READDRIVESTATUS***********************)
	MC_BR_ReadDriveStatus_0.Enable := NOT(MC_BR_ReadDriveStatus_0.Error);
	MC_BR_ReadDriveStatus_0.Axis := AxisREF;
	MC_BR_ReadDriveStatus_0.AdrDriveStatus := ADR(BasicControl.Status.DriveStatus);
	MC_BR_ReadDriveStatus_0();
	(************************ MC_READSTATUS *************************)
	MC_ReadStatus_0.Enable :=  NOT MC_ReadStatus_0.Error;
	MC_ReadStatus_0.Axis := AxisREF;
	MC_ReadStatus_0();

	//**********	diameter estimation	top winder	******************
	MC_ReadActualPosition_0.Axis 	:= AxisREF;
	MC_ReadActualPosition_0.Enable 	:= TRUE;
	MC_ReadActualPosition_0();
	MC_ReadActualVelocity_0.Axis 	:= AxisREF;
	MC_ReadActualVelocity_0.Enable	:= TRUE;
	MC_ReadActualVelocity_0();
	machineaxis.MC_ReadActualPosition_0();
	machineaxis.MC_ReadActualVelocity_0();
	WNCCalcDiam_0.enable			:= TRUE;
	WNCCalcDiam_0.startDiam 		:= startdiameter; // estimation of start diameter in [mm]

	WNCCalcDiam_0.actLinePos		:=  pMasteraxisREF.monitor.s; // gMaster1.monitor.s;
	//	WNCCalcDiam_0.actLinePos		:= REAL_TO_DINT (machineaxis.MC_ReadActualPosition_0.Position); (*( masteraxisREF.monitor.s);*)
	//	WNCCalcDiam_0.actLineSpeed		:=  machineaxis.MC_ReadActualVelocity_0.Velocity;
	WNCCalcDiam_0.actLineSpeed		:= pMasteraxisREF.monitor.v;
	IF data.recipeData.reverse (*AND NOT  MC_TorqueControl_0.Active*) AND data.machData.axistyp = 1 THEN
		(*	WNCCalcDiam_0.actWndPos		:=  REAL_TO_DINT (MC_ReadActualPosition_0.Position); // gTWindTop.monitor.s;*)
		WNCCalcDiam_0.actWndPos		:= pAxis.monitor.s; //06.03.15
		WNCCalcDiam_0.actWndSpeed	:= MC_ReadActualVelocity_0.Velocity;
	ELSIF NOT data.recipeData.reverse (*AND NOT  MC_TorqueControl_0.Active*)  AND data.machData.axistyp = 1 THEN
		(*	WNCCalcDiam_0.actWndPos		:= - REAL_TO_DINT (MC_ReadActualPosition_0.Position); /*)// gTWindTop.monitor.s;
		WNCCalcDiam_0.actWndPos		:= - pAxis.monitor.s; //06.03.15
		WNCCalcDiam_0.actWndSpeed	:= -MC_ReadActualVelocity_0.Velocity;
	END_IF
	IF data.recipeData.reverse AND data.machData.axistyp = - 1 THEN
		(*WNCCalcDiam_0.actWndPos		:= -REAL_TO_DINT (MC_ReadActualPosition_0.Position);*) // gTWindTop.monitor.s;
		WNCCalcDiam_0.actWndPos		:= - pAxis.monitor.s; //06.03.15
	ELSIF NOT data.recipeData.reverse AND data.machData.axistyp = - 1 THEN
		(*WNCCalcDiam_0.actWndPos		:= REAL_TO_DINT (MC_ReadActualPosition_0.Position);*) // gTWindTop.monitor.s;
		WNCCalcDiam_0.actWndPos		:=  pAxis.monitor.s; //06.03.15
	END_IF

	IF machineaxis.MC_ReadStatus_0.ContinuousMotion THEN (*anhalten des Durchmesserrechners*)
		WNCCalcDiam_0.hold := FALSE;
	ELSE
		WNCCalcDiam_0.hold := TRUE;
	END_IF
	WNCCalcDiam_0.mode			:= 1;(*1 = Position 2 = Speed*)
//	WNCCalcDiam_0.setStartDiam	:= TRUE; // gMachine.Status.mManualModeActive;
	WNCCalcDiam_0();

	LCRLimit_0.min_value				:= 90;
	LCRLimit_0.max_value				:= 600;
	LCRLimit_0.in						:= WNCCalcDiam_0.actDiam;
	LCRLimit_0();

	//************************* Bahnrissüberwachung *******************
	IF machineaxis.MC_ReadStatus_0.StandStill THEN
		IF  merker THEN
			test1 :=  fmod(MC_ReadActualPosition_0.Position,DINT_TO_REAL (LCRLimit_0.out));
			merker := FALSE;
		END_IF
		IF 	test1 < fmod(MC_ReadActualPosition_0.Position,DINT_TO_REAL (LCRLimit_0.out)) THEN
//	 		MC_TorqueControl_0.Execute := FALSE;
		END_IF
	ELSIF machineaxis.MC_ReadStatus_0.ContinuousMotion THEN
			merker := TRUE;
	END_IF
	//*****************************************************************

	TC_Winder_0.ActDiameter				:= LCRLimit_0.out * SCALE_MM_TO_DRIVE_UNITS; // gMachine.Status.Diam.TUnwindTop * SCALE_MM_TO_DRIVE_UNITS;
	TC_Winder_0.EncoderIf				:= pAxis.encoder_if.parameter; // gTWindTop.encoder_if.parameter;
	TC_Winder_0.GearRatio				:= data.machData.GEAR_RATIO;
	TC_Winder_0.LineUnits				:= MACHINE_UNITS_PER_METER;
	//	TC_Winder_0.SetLineSpeed			:= machineaxis.MC_ReadActualVelocity_0.Velocity; (*machineaxis.velocity;*)  //AxisIf.Status.ActMasterVelocity;
	TC_Winder_0.SetLineSpeed			:= pMasteraxisREF.monitor.v;//23.03.15
	TC_Winder_0.RefDiameter[0]			:= data.machData.coreDiam; //gApplRecipe.endModule.minDiamValueTop;
//	TC_Winder_0.RefDiameter[1]			:= data.machData.stopDiam * SCALE_MM_TO_DRIVE_UNITS;//gMachRecipe.topTandemWind.StopDiam * SCALE_MM_TO_DRIVE_UNITS;
	TC_Winder_0.RefTension[0]			:= LIMIT(0, data.recipeData.minDiamTension, 80); // gApplRecipe.endModule.minDiamTensionTop;
	TC_Winder_0.RefTension[1]			:= LIMIT (0, data.recipeData.maxDiamTension, 80); //gApplRecipe.endModule.maxDiamTensionTop;
	TC_Winder_0();

	// Reduzierung des Momentes zum hoch und runterfahren des

	IF NOT mode THEN (* reduzierung des Moments damit der Bahnspeicher nach oben (Füllen) fahren kann*)
		IF data.recipeData.reverse(* AND NOT  MC_TorqueControl_0.Active*) THEN
			settorque	:= LIMIT(-80, -1 * (TC_Winder_0.SetMotorTorque + data.machData.frictionCompensation), 0);
		ELSE
			settorque	:= LIMIT (0, TC_Winder_0.SetMotorTorque + data.machData.frictionCompensation, 80);
		END_IF;
	ELSE
		IF data.recipeData.reverse  (*AND NOT  MC_TorqueControl_0.Active*) THEN
			settorque	:= LIMIT(-80, (-1 * TC_Winder_0.SetMotorTorque) + torqueoffset, 0);
		ELSE
			settorque	:= LIMIT (0, TC_Winder_0.SetMotorTorque - torqueoffset, 80);
		END_IF;
	END_IF

	// Reduzierung des Momentes zum hoch und runterfahren des // OKrebs 16.09.14
	IF	bufferUpDownKeys THEN
		IF data.recipeData.reverse  (*AND NOT  MC_TorqueControl_0.Active*) THEN
			settorque	:= LIMIT(-80, (-1 * TC_Winder_0.SetMotorTorque) + torqueoffset, 0);
		ELSE
			settorque	:= LIMIT (0, TC_Winder_0.SetMotorTorque - torqueoffset, 80);
		END_IF;
	END_IF
	//////////

	MC_TorqueControl_0.Velocity	:= TC_Winder_0.SetWndSpeed * ( 102/ 100.0) (*AxisIf.Para.WinderVeloOffsetHz*data.machData.velocityOverride  *);
	IF ABS (MC_TorqueControl_0.Torque) <> ABS (settorque) (*AND data.recipeData.mode = CONST.UNITMODEs.ENABLE*) THEN (* wenn das Moment sich aendert muss Exucute weg genommen werden*)
		MC_TorqueControl_0.Execute := FALSE;
		cmd := CONST.AXIS.START;
		enablemerker := TRUE;
	END_IF

	MC_TorqueControl_0.TorqueRamp := 10;
	MC_TorqueControl_0.Acceleration := 20000;
	MC_TorqueControl_0.Axis		:= AxisREF;
 	MC_TorqueControl_0.Torque	:= settorque;
(*	MC_TorqueControl_0();*)
	IF 	(cmd = CONST.AXIS.START AND NOT MC_TorqueControl_0.InTorque )AND (MC_ReadStatus_0.StandStill OR MC_ReadStatus_0.ContinuousMotion) THEN
		(*MC_Stop_0.Execute := FALSE*);
		MC_TorqueControl_0.Execute := TRUE;
		cmdtmp := cmd;
		cmd:= CONST.AXIS.NOACTION;
	END_IF
	IF MC_TorqueControl_0.Execute AND MC_TorqueControl_0.CommandAborted AND cmdtmp = CONST.AXIS.START THEN
		MC_TorqueControl_0.Execute := FALSE;
//	ELSIF NOT MC_TorqueControl_0.Execute  AND cmdtmp = CONST.AXIS.POWER_ON AND NOT MC_TorqueControl_0.Error AND MC_ReadStatus_0.StandStill THEN
//		MC_TorqueControl_0.Execute := TRUE;
	END_IF
	MC_TorqueControl_0();
//	IF enablemerker (*AND NOT MC_TorqueControl_0.Active*) THEN
//		MC_TorqueControl_0.Execute := TRUE;(*wieder einschalten*)
//		enablemerker := FALSE;
//	END_IF
	IF cmd = CONST.AXIS.POWER_ON THEN
		MC_Power_0.Enable := TRUE;
		IF MC_Power_0.Status THEN
			cmdtmp := cmd;
			WNCCalcDiam_0.setStartDiam 		:= TRUE; // set startDiam when FB is enabled
			cmd := CONST.AXIS.NOACTION;
		END_IF
	ELSIF cmd = CONST.AXIS.POWER_OFF THEN
		MC_Power_0.Enable := FALSE;
		MC_TorqueControl_0.Execute := FALSE;
		IF NOT MC_Power_0.Status THEN
			cmdtmp := cmd;
			WNCCalcDiam_0.setStartDiam 		:= FALSE; // set startDiam when FB is enabled
			cmd:= CONST.AXIS.NOACTION;
		END_IF
	ELSIF cmd = CONST.AXIS.RESET THEN
		MC_Stop_0.Execute := FALSE;
		MC_Power_0.Enable := FALSE;
		MC_Reset_0.Execute := TRUE;
		IF MC_Reset_0.Done THEN
			MC_Reset_0.Execute := FALSE;
			cmdtmp := cmd;
			cmd:= CONST.AXIS.NOACTION;
		END_IF

	END_IF
	MC_Stop_0.Deceleration	:= deceleration;
	IF cmd = CONST.AXIS.STOP THEN
		IF  MC_ReadStatus_0.ContinuousMotion OR MC_ReadStatus_0.DiscreteMotion
			OR MC_ReadStatus_0.SynchronizedMotion THEN
				MC_TorqueControl_0.Execute := FALSE;
				MC_Stop_0.Execute := TRUE;
		END_IF
		IF MC_Stop_0.Done THEN
			MC_Stop_0.Execute := FALSE;
			cmdtmp := cmd;
			cmd := CONST.AXIS.NOACTION;
		END_IF
	END_IF
	(***************************************************************
        FUNCTION Block Calls
	(************************** MC_STOP *****************************)
	MC_Stop_0.Axis := AxisREF;
	MC_Stop_0();
	(************************** MC_POWER ****************************)
	MC_Power_0.Axis := AxisREF;  (* pointer to axis *)
	MC_Power_0();
	(************************** MC_RESET ****************************)
	MC_Reset_0.Axis := AxisREF;
	MC_Reset_0();
END_FUNCTION_BLOCK
```

#### ac_setStateAfterWinder.st
```iecst
(********************************************************************
 * COPYRIGHT -- Microsoft
 ********************************************************************
 * Programm: MAIN
 * Datei: ac_setStateAfterUnwinder.st
 * Autor: Awalz
 * Erstellt: 7. April 2014
 ********************************************************************
 * Implementierung des Programms MAIN
 ********************************************************************)

 (*<$Description$> Fügt eine neue Aktion zum IEC Programm oder Bibliothek </$Description$>*)
ACTION ac_setStateAfterWinder:
	IF BetrCtrl.value = CONST.MACHINEMODES.EMERGENCYSTOP THEN
		StateCtrl := CTRL_EMERGENCYSTOP_BEFORE;
	ELSIF BetrCtrl.value = CONST.MACHINEMODES.SAFETYSTOP THEN
		StateCtrl := CTRL_SAFETYSTOP_BEFORE;
	ELSIF BetrCtrl.value = CONST.MACHINEMODES.MANUAL THEN
		StateCtrl := CTRL_STOP_BEFORE;
	ELSIF BetrCtrl.value = CONST.MACHINEMODES.AUTOMATIC THEN
		StateCtrl := CTRL_STOP_BEFORE;
	END_IF
END_ACTION
```

#### ac_manualWinder.st
```iecst
(********************************************************************
 * COPYRIGHT -- Microsoft
 ********************************************************************
 * Programm: MAIN
 * Datei: ac_manualUnwinder.st
 * Autor: Awalz
 * Erstellt: 7. April 2014
 ********************************************************************
 * Implementierung des Programms MAIN
 ********************************************************************)

 (*<$Description$> Fügt eine neue Aktion zum IEC Programm oder Bibliothek </$Description$>*)
ACTION ac_manualWinder:
		CASE state OF
	ST_IDLE:
		IF BetrCtrl.value <> CONST.MACHINEMODES.MANUAL THEN
			state := ST_IDLE;
			err(reset := TRUE);
			busy := TRUE;
			status.ready := FALSE;
			StateCtrl := CTRL_MANUAL_AFTER;
		ELSE
			IF data.recipeData.mode = CONST.UNITMODEs.ENABLE AND NOT winderaxis.MC_TorqueControl_0.Error THEN
				winderaxis.cmd := CONST.AXIS.START;
			ELSE
				winderaxis.cmd := CONST.AXIS.STOP;
			END_IF
		(*	ButtonUp.lamp.aktion := SEL(unwinder.aushub.isup OR ButtonUp.key.inp, CONST.LAMP.OFF, CONST.LAMP.ON);
			ButtonDown.lamp.aktion := SEL(unwinder.aushub.isdown OR ButtonDown.key.inp, CONST.LAMP.OFF, CONST.LAMP.ON);
			unwinder.aushub.manual(
				buttonUP 	:=  ButtonUp.key.inp
									AND NOT unwinder.aushub.isup,
				buttonDown 	:=  ButtonDown.key.inp
									AND NOT unwinder.aushub.isdown);
(*			unwinder.brake.control(dancer := dancer, radius := unwinder.radius); *)
		(*	webGuidng.manual();
			unwinder.ctrl(cmd := unwinder.ctrl.cmdVISU, brake := unwinder.brake, aushub := unwinder.aushub, radius := unwinder.radius, dancer := dancer, status := unwinder.status, data := unwinder.data, machineMaster := machineMaster);
(*			status.ready := unwinder.status.ready; *)
		END_IF
	END_CASE
END_ACTION
```

#### Package Logical/MainMachineCtrl/MAIN/PackBelt - Paket

#### FB_PackBelt.st
```iecst
(********************************************************************
 * COPYRIGHT -- Microsoft
 ********************************************************************
 * Programm: MAIN
 * Datei: FB_PackBelt.st
 * Autor: okrebs
 * Erstellt: 23. November 2016
 ********************************************************************
 * Implementierung des Programms MAIN
 ********************************************************************)

(* TODO: Bitte Kommentar hier einfügen *)
FUNCTION_BLOCK FB_PackBelt
END_FUNCTION_BLOCK
```

#### FB_PackBeltCtrl.st
```iecst
(********************************************************************
 * COPYRIGHT -- Microsoft
 ********************************************************************
 * Programm: MAIN
 * Datei: FB_PackBeltCtrl.st
 * Autor: okrebs
 * Erstellt: 23. November 2016
 ********************************************************************
 * Implementierung des Programms MAIN
 ********************************************************************)

(* TODO: Bitte Kommentar hier einfügen *)
FUNCTION_BLOCK FB_PackBeltCtrl

	PackBelt_HW;
	PackBelt_DrvIf;
	PackBelt_DiDoIf;

	// Initialisation
	IF firststart THEN
		pAxis ACCESS axisREF;

		MC_BR_JogVelocity_0.Axis := axisREF;
		MC_Power_0.Axis := axisREF;
		MC_Stop_0.Axis := axisREF;
		MC_Reset_0.Axis := axisREF;
		MC_ReadStatus_0.Axis := axisREF;
		Time_Conveyor_To_Box_s := 2;
		Range_Conveyor_To_Box := 200000;  // vorher 300000 // OKrebs // 09.09.21

		firststart := FALSE;
	END_IF

	MC_ReadStatus_0.Enable :=  NOT MC_ReadStatus_0.Error;
	MC_BR_JogVelocity_0.Acceleration	:= data.acceleration;
	MC_BR_JogVelocity_0.Deceleration	:= data.deceleration;
	TP_PowerOn(IN := Start_TP_PowerOn, PT := T#100ms); // Zeit um den Motor einzuschalten
	IF conveyor.axis.ctrl.MC_ReadActualVelocity_0.Velocity > 0 AND MC_ReadStatus_0.ContinuousMotion THEN
		Time_Conveyor_To_Box_s := (masterModul.data.periodLength + Range_Conveyor_To_Box) / conveyor.axis.ctrl.MC_ReadActualVelocity_0.Velocity; // Zeit bis der letzte Stanzling in die Box fällt
	END_IF
//	TON_Nitto_Table_Full(IN := conveyor.counters.Nitto_Table_Full, PT := REAL_TO_TIME(Time_Conveyor_To_Box_s * 1000));
	TON_Nitto_Table_Full(IN := conveyor.counters.Nitto_Table_Full, PT := T#200ms); // vorher 500ms // OKrebs // 09.09.21
	Start_TP_PowerOn := FALSE;

	R_TRIG_NittoTableFull(CLK := TON_Nitto_Table_Full.Q);
	R_TRIG_LowerSpeed(CLK := sensorLowerSpeed OR testLowerSpeed);
	R_TRIG_Stop(CLK := sensorStop OR TestStop);

	// 24.07.18 // OKrebs // Resetfunktion
	IF panel.LDTRESET.LDT.button AND (MC_ReadStatus_0.Error OR MC_ReadStatus_0.Errorstop)  THEN
		MC_Reset_0.Execute := TRUE;
		state := ST_WAIT;
	END_IF
	/////////////////////

	/////////////////////////////////////STEUERUNG/////////////////////////////////////////////
	CASE state OF

		ST_WAIT:
			IF (switchAutomatic AND R_TRIG_NittoTableFull.Q AND NOT sensorBoxesPresent) OR
				(switchManual AND buttonStart AND NOT sensorBoxesPresent) THEN
				MC_Power_0.Enable := TRUE;
				Start_TP_PowerOn := TRUE;
			END_IF

			IF NOT TP_PowerOn.Q AND MC_ReadStatus_0.StandStill THEN
				MC_BR_JogVelocity_0.Velocity := data.highSpeed;
				MC_BR_JogVelocity_0.Enable := TRUE;
				MC_BR_JogVelocity_0.JogPositive := TRUE;
				state := ST_MOVE_FAST;
			END_IF

		ST_MOVE_FAST:
			IF R_TRIG_LowerSpeed.Q THEN
				MC_BR_JogVelocity_0.Velocity := data.lowSpeed;
				state := ST_MOVE_SLOW;
			END_IF

		ST_MOVE_SLOW:
			IF R_TRIG_Stop.Q THEN
				MC_BR_JogVelocity_0.JogPositive := FALSE;
				MC_BR_JogVelocity_0.Enable := FALSE;
			END_IF

			IF MC_ReadStatus_0.StandStill THEN
				MC_Power_0.Enable := FALSE;
			END_IF

			IF MC_ReadStatus_0.Disabled THEN
				state := ST_WAIT;
			END_IF

	END_CASE

	///////////////////////////////////////////////////////////////////////////////////////////

	MC_ReadStatus_0();
	MC_Reset_0();
	MC_Power_0();
	MC_Stop_0();
	MC_BR_JogVelocity_0();

END_FUNCTION_BLOCK
```
